// TwinCAT 3 PLC project Master_0000_Allgemein
// ProgramVersion: 3.1.4026.20
// libraries:
//   BASIC, * (OSCAT)
//   Tc2_EtherCAT, * (Beckhoff Automation GmbH)
//   Tc2_MC2, * (Beckhoff Automation GmbH)
//   Tc2_MC2_Drive, * (Beckhoff Automation GmbH)
//   Tc2_NC, * (Beckhoff Automation GmbH)
//   Tc2_Standard, * (Beckhoff Automation GmbH)
//   Tc2_System, * (Beckhoff Automation GmbH)
//   Tc2_Utilities, * (Beckhoff Automation GmbH)
//   Tc3_Database, * (Beckhoff Automation GmbH)
// project tree:
//   0000/ Ablauf_0000.TcPOU, EAs_0000.TcGVL (not stored), GVL_0000.TcGVL (not stored), GVL_Meldungen.TcGVL (not stored), GVL_Visu_0000.TcGVL, Hardware_0000.TcPOU (not stored)
//   1000_Allgemein/ Ablauf_1000.TcPOU (not stored), EAs_1000.TcGVL, GVL_1000.TcGVL, GVL_Visu_1000.TcGVL, Hardware_1000.TcPOU (not stored)
//   3100_Bohraggregat/ Ablauf_3100.TcPOU, EAs_3100.TcGVL (not stored), GVL_3100.TcGVL (not stored), GVL_Visu_3100.TcGVL, Hardware_3100.TcPOU (not stored)
//   3200_Bohraggregat/ Ablauf_3200.TcPOU (not stored), EAs_3200.TcGVL (not stored), GVL_3200.TcGVL, GVL_Visu_3200.TcGVL, Hardware_3200.TcPOU (not stored)
//   3300_Bohraggregat/ Ablauf_3300.TcPOU, EAs_3300.TcGVL, GVL_3300.TcGVL (not stored), GVL_Visu_3300.TcGVL, Hardware_3300.TcPOU
//   3400_Bohraggregat/ Ablauf_3400.TcPOU (not stored), EAs_3400.TcGVL, GVL_3400.TcGVL, GVL_Visu_3400.TcGVL (not stored), Hardware_3400.TcPOU
//   3510_Transport/ Ablauf_3510.TcPOU, EAs_3510.TcGVL (not stored), GVL_3510.TcGVL, GVL_Visu_3510.TcGVL (not stored), Hardware_3510.TcPOU
//   3520_Transport/ Ablauf_3520.TcPOU, EAs_3520.TcGVL (not stored), GVL_3520.TcGVL, GVL_Visu_3520.TcGVL, Hardware_3520.TcPOU (not stored)
//   3530_Niederhalter/ Ablauf_3530.TcPOU, EAs_3530.TcGVL (not stored), GVL_3530.TcGVL, GVL_Visu_3530.TcGVL (not stored), Hardware_3530.TcPOU (not stored)
//   3540_Niederhalter/ Ablauf_3540.TcPOU, EAs_3540.TcGVL, GVL_3540.TcGVL (not stored), GVL_Visu_3540.TcGVL (not stored), Hardware_3540.TcPOU
//   / MAIN.TcPOU (not stored), PlcTask.TcTTO (not stored)
//   SRT_Allgemein/0010_Bausteine_mitDuts/Blink/ GVL_Blink.TcGVL (not stored), PRG_Blink.TcPOU (not stored)
//   SRT_Allgemein/0010_Bausteine_mitDuts/DUTs/ DUT_Visu_SteuerStatus.TcDUT
//   SRT_Allgemein/0010_Bausteine_mitDuts/DUTs/Meldungen/ DUT_Diagnose_1000.TcDUT (not stored), DUT_Diagnose_2000.TcDUT (not stored), DUT_Diagnose_3000.TcDUT, DUT_Diagnose_4000.TcDUT, DUT_Diagnose_5000.TcDUT, DUT_Meldungen_0000.TcDUT, DUT_Diagnose_0000.TcDUT (not stored), DUT_Meldungen_1000.TcDUT, DUT_Meldungen_2000.TcDUT, DUT_Meldungen_3000.TcDUT (not stored), DUT_Meldungen_4000.TcDUT, DUT_Meldungen_5000.TcDUT
//   SRT_Allgemein/0010_Bausteine_mitDuts/DUTs/Rexroth FU/ DUT_Rexroth_FU_PD_IN.TcDUT (not stored), DUT_Rexroth_FU_PD_OUT.TcDUT (not stored), DUT_Rexroth_FU_steuern.TcDUT
//   SRT_Allgemein/0010_Bausteine_mitDuts/DUTs/Safety/ DUT_EL1918_Logic.TcDUT (not stored), E_ModeLanguage.TcDUT (not stored), ST_InfoDataConnection_1904.TcDUT (not stored), ST_InfoDataConnection_1918.TcDUT, ST_InfoDataFB.TcDUT (not stored), ST_InfoDataGroup.TcDUT (not stored)
//   SRT_Allgemein/0010_Bausteine_mitDuts/DUTs/Servo/ DUT_Achse_koppeln.TcDUT (not stored), DUT_Achse_Service.TcDUT, DUT_Achse_Status.TcDUT, DUT_Achse_Steuern.TcDUT (not stored), DUT_Geschwindigkeitsabgleich.TcDUT (not stored), DUT_NC_Kanal.TcDUT (not stored), DUT_PD_InOut_Achsen.TcDUT, DUT_Rexroth_Parameter.TcDUT
//   SRT_Allgemein/0010_Bausteine_mitDuts/DUTs/SEW_Movitrac/COE/ st_COE_Parameter.TcDUT, st_COE_Parameter_Out.TcDUT (not stored)
//   SRT_Allgemein/0010_Bausteine_mitDuts/DUTs/SEW_Movitrac/CSV_BASE/ st_CSV_Database.TcDUT (not stored), st_MaschParameter.TcDUT (not stored)
//   SRT_Allgemein/0010_Bausteine_mitDuts/DUTs/SEW_Movitrac/ DUT_SEW_FU_PD_IN.TcDUT (not stored), DUT_SEW_FU_PD_OUT.TcDUT (not stored), DUT_SEW_FU_Status.TcDUT, DUT_SEW_FU_Steuern.TcDUT (not stored), DUT_SEW_FU_Visu.TcDUT, DUT_SEW_Para.TcDUT (not stored)
//   SRT_Allgemein/0010_Bausteine_mitDuts/DUTs/Ventil/ DUT_Ventil_para.TcDUT, DUT_Ventil_sps.TcDUT (not stored), DUT_Ventil_VISU.TcDUT, DUT_VorZur_visu.TcDUT (not stored)
//   SRT_Allgemein/0010_Bausteine_mitDuts/POUs/ FB_Achs_Freigabe.TcPOU, FB_Anst_Vakuum.TcPOU (not stored), FB_Automatik.TcPOU, FB_Belegt.TcPOU, FB_Bereichsueberwachung.TcPOU, FB_FuStart_Fraese.TcPOU (not stored), FB_FU_Rexroth.TcPOU, FB_inRange.TcPOU (not stored), FB_Kollision.TcPOU (not stored), FB_Messachse_EL3051.TcPOU, FB_Messachse_EL5151.TcPOU (not stored), FB_Messauswertung_Hysterese.TcPOU (not stored), FB_normieren.TcPOU (not stored), FB_PneuPosition.TcPOU (not stored), FB_Schutztuer_mitBremsentest.TcPOU, FB_Toggle_Anforderung.TcPOU (not stored), FB_Toogle.TcPOU (not stored), FB_Transport.TcPOU (not stored), FB_Umrechnung.TcPOU (not stored), FB_Ventil.TcPOU, FB_Ventil_V2.TcPOU, FC_Bereichsueberwachung.TcPOU, FC_InRange.TcPOU, Func_InRange.TcPOU (not stored), IBN_Huettenhoelscher.TcPOU (not stored)
//   SRT_Allgemein/0010_Bausteine_mitDuts/POUs/FU_SEW/Movi_B/ FB_SEW_MOVITRAC.TcPOU, FB_SEW_MOVITRAC_CoE.TcPOU (not stored)
//   SRT_Allgemein/0010_Bausteine_mitDuts/POUs/FU_SEW/Movi_C/ FB_SEW_MOVITRAC_C_COE.TcPOU, FB_SEW_MOVITRAC_C_COE_18000Umin.TcPOU (not stored)
//   SRT_Allgemein/0010_Bausteine_mitDuts/POUs/FU_SEW/sub/CoE/ fb_CoeDataRead.TcPOU (not stored), fb_CoeDataWrite.TcPOU (not stored)
//   SRT_Allgemein/0010_Bausteine_mitDuts/POUs/FU_SEW/sub/CSV Read_Write/ fb_CSVBaseRead.TcPOU, fb_CSVBaseWrite.TcPOU (not stored), fb_OrdnerErstellen.TcPOU, fb_Parameter_CSV.TcPOU
//   SRT_Allgemein/0010_Bausteine_mitDuts/POUs/FU_SEW/sub/ FB_SEW_CoE.TcPOU (not stored)
//   SRT_Allgemein/0010_Bausteine_mitDuts/POUs/Safety/ FB_InfoConnection_1904.TcPOU (not stored), FB_InfoConnection_1918.TcPOU, FB_InfoEStop.TcPOU, FB_InfoGroup.TcPOU (not stored)
//   SRT_Allgemein/0010_Bausteine_mitDuts/POUs/Servos_NC/ FB_Achse_NC_PTP_Beckhoff.TcPOU (not stored), FB_Achse_NC_PTP_Master_Slave_v2.TcPOU, FB_Achse_NC_PTP_V3.TcPOU, FB_Achse_NC_PTP_V4.TcPOU, FB_Achse_NC_PTP_V4_1.TcPOU (not stored), FB_Achse_NC_PTP_V4_2.TcPOU, FB_Achse_NC_PTP_Velo.TcPOU (not stored), FB_MasterSlaveSpeedControl.TcPOU, FB_Nc_Kanal.TcPOU, Rexroth_Servo_Modulo.TcPOU (not stored)
//   SRT_Allgemein/0010_Bausteine_mitDuts/POUs/Zaehler/ FB_Laufzeit.TcPOU, FB_SpindelInBearbeitung.TcPOU
//   SRT_Allgemein/Bus/ Busdiagnose.TcPOU, DUT_Busdiagnose.TcDUT, DUT_Busdiagnose_Daten.TcDUT (not stored), GVL_Busdiagnose.TcGVL (not stored)
// real-time tasks:
//   TASK PlcTask: cycle T#10ms, priority 20, ADS port 350
// motion (NC):
//   TASK NC-Task 1 SAF: cycle T#2ms, priority 4, ADS port 501
//   TASK NC-Task 1 SVB: cycle T#10ms, priority 8, ADS port 511
//   AXIS =3100+FS2-11M1 (X-Achse) (id 1)
//     OtherSettings: AllowMotionCmdToSlave=true
//     encoder EncType=19
//       EncPara: MaxCount=#xffffffff
//     drive DrvType=16
//       DrvPara: MaxCount=#xffffffff
//         Analog: TorqueSetpointScale=10, ScaleFactorActTorque=0.1
//         TimeComp: TaskDelayCycles=1
//     controller CtrType=1
//       CtrPara: PriorControlFactor=1
//         Observer: BandWidth=20
//   AXIS =3100+FS2-12M1 (Y-Achse) (id 2)
//     OtherSettings: AllowMotionCmdToSlave=true
//     encoder EncType=19
//       EncPara: MaxCount=#xffffffff
//     drive DrvType=16
//       DrvPara: MaxCount=#xffffffff
//         Analog: TorqueSetpointScale=10, ScaleFactorActTorque=0.1
//         TimeComp: TaskDelayCycles=1
//     controller CtrType=1
//       CtrPara: PriorControlFactor=1
//         Observer: BandWidth=20
//   AXIS =3100+FS2-13M1 (Z-Achse) (id 3)
//     OtherSettings: AllowMotionCmdToSlave=true
//     encoder EncType=19
//       EncPara: MaxCount=#xffffffff
//     drive DrvType=16
//       DrvPara: MaxCount=#xffffffff
//         Analog: TorqueSetpointScale=10, ScaleFactorActTorque=0.1
//         TimeComp: TaskDelayCycles=1
//     controller CtrType=1
//       CtrPara: PriorControlFactor=1
//         Observer: BandWidth=20
//   AXIS =3200+FS2-11M1 (X-Achse) (id 4)
//     OtherSettings: AllowMotionCmdToSlave=true
//     encoder EncType=19
//       EncPara: MaxCount=#xffffffff
//     drive DrvType=16
//       DrvPara: MaxCount=#xffffffff
//         Analog: TorqueSetpointScale=10, ScaleFactorActTorque=0.1
//         TimeComp: TaskDelayCycles=1
//     controller CtrType=1
//       CtrPara: PriorControlFactor=1
//         Observer: BandWidth=20
//   AXIS =3200+FS2-12M1 (Y-Achse) (id 5)
//     OtherSettings: AllowMotionCmdToSlave=true
//     encoder EncType=19
//       EncPara: MaxCount=#xffffffff
//     drive DrvType=16
//       DrvPara: MaxCount=#xffffffff
//         Analog: TorqueSetpointScale=10, ScaleFactorActTorque=0.1
//         TimeComp: TaskDelayCycles=1
//     controller CtrType=1
//       CtrPara: PriorControlFactor=1
//         Observer: BandWidth=20
//   AXIS =3200+FS2-13M1 (Z-Achse) (id 6)
//     OtherSettings: AllowMotionCmdToSlave=true
//     encoder EncType=19
//       EncPara: MaxCount=#xffffffff
//     drive DrvType=16
//       DrvPara: MaxCount=#xffffffff
//         Analog: TorqueSetpointScale=10, ScaleFactorActTorque=0.1
//         TimeComp: TaskDelayCycles=1
//     controller CtrType=1
//       CtrPara: PriorControlFactor=1
//         Observer: BandWidth=20
//   AXIS =3300+FS2-11M1 (X-Achse) (id 7)
//     OtherSettings: AllowMotionCmdToSlave=true
//     encoder EncType=19
//       EncPara: MaxCount=#xffffffff
//     drive DrvType=16
//       DrvPara: MaxCount=#xffffffff
//         Analog: TorqueSetpointScale=10, ScaleFactorActTorque=0.1
//         TimeComp: TaskDelayCycles=1
//     controller CtrType=1
//       CtrPara: PriorControlFactor=1
//         Observer: BandWidth=20
//   AXIS =3300+FS2-12M1 (Y-Achse) (id 8)
//     OtherSettings: AllowMotionCmdToSlave=true
//     encoder EncType=19
//       EncPara: MaxCount=#xffffffff
//     drive DrvType=16
//       DrvPara: MaxCount=#xffffffff
//         Analog: TorqueSetpointScale=10, ScaleFactorActTorque=0.1
//         TimeComp: TaskDelayCycles=1
//     controller CtrType=1
//       CtrPara: PriorControlFactor=1
//         Observer: BandWidth=20
//   AXIS =3400+FS2-11M1 (X-Achse) (id 9)
//     OtherSettings: AllowMotionCmdToSlave=true
//     encoder EncType=19
//       EncPara: MaxCount=#xffffffff
//     drive DrvType=16
//       DrvPara: MaxCount=#xffffffff
//         Analog: TorqueSetpointScale=10, ScaleFactorActTorque=0.1
//         TimeComp: TaskDelayCycles=1
//     controller CtrType=1
//       CtrPara: PriorControlFactor=1
//         Observer: BandWidth=20
//   AXIS =3400+FS2-12M1 (Y-Achse) (id 10)
//     OtherSettings: AllowMotionCmdToSlave=true
//     encoder EncType=19
//       EncPara: MaxCount=#xffffffff
//     drive DrvType=16
//       DrvPara: MaxCount=#xffffffff
//         Analog: TorqueSetpointScale=10, ScaleFactorActTorque=0.1
//         TimeComp: TaskDelayCycles=1
//     controller CtrType=1
//       CtrPara: PriorControlFactor=1
//         Observer: BandWidth=20
//   AXIS =3520+FS2-11M1 (Y-Achse) (id 11)
//     OtherSettings: AllowMotionCmdToSlave=true
//     encoder EncType=19
//       EncPara: MaxCount=#xffffffff
//     drive DrvType=16
//       DrvPara: MaxCount=#xffffffff
//         Analog: TorqueSetpointScale=10, ScaleFactorActTorque=0.1
//         TimeComp: TaskDelayCycles=1
//     controller CtrType=1
//       CtrPara: PriorControlFactor=1
//         Observer: BandWidth=20
//   AXIS =3540+FS2-11M1 (Y-Achse) (id 12)
//     OtherSettings: AllowMotionCmdToSlave=true
//     encoder EncType=19
//       EncPara: MaxCount=#xffffffff
//     drive DrvType=16
//       DrvPara: MaxCount=#xffffffff
//         Analog: TorqueSetpointScale=10, ScaleFactorActTorque=0.1
//         TimeComp: TaskDelayCycles=1
//     controller CtrType=1
//       CtrPara: PriorControlFactor=1
//         Observer: BandWidth=20
// I/O:
//   DEVICE Gerät 1 (EtherCAT), AmsNetId 169.254.68.135.2.1
//     +FS1-3K1 (BK1120) [EK1100 EtherCAT-Koppler (2A E-Bus)]
//       +FS1-3K2 (EL6070-0033) [EL6070-0033 1K. Licence-Key-Klemme, individuelle Lizenzen]
//       +FS1-3K3 (EL1918) [EL1918, 8K. Safety Eingang 24V, TwinSAFE]
//         modules: Module 1 (FSOE), Module 2 (FSLOGIC)
//       +FS1-3K4 (EL2904) [EL2904, 4 K. Safety Ausgang 24V, 0.5A, TwinSAFE]
//         modules: Module 1 (FSOES), Module 2 (DO)
//       +FS1-3K5 (EL1809)
//       +FS1-3K6 (EL2809)
//       +FS1-3A1 (EL9011)
//     +K110-1K1 (BK1120)
//     =3100+FS2-16T1 (Bohraggr Schlosskastenfräser) [MOVI-C MOVITRAC]
//       modules: Module 1 (Standard 16 PD)
//     =3100+FS2-17T1 (Bohraggr Vorbohren) [MOVI-C MOVITRAC]
//       modules: Module 1 (Standard 16 PD)
//     =3100+FS2-18T1 (Bohraggr Stulpfräser) [MOVI-C MOVITRAC]
//       modules: Module 1 (Standard 16 PD)
//     =3200+FS2-16T1 (Bohraggr Stufenbohrer) [MOVI-C MOVITRAC]
//       modules: Module 1 (Standard 16 PD)
//     =3200+FS2-17T1 (Bohraggr Stulpfräser) [MOVI-C MOVITRAC]
//       modules: Module 1 (Standard 16 PD)
//     =3300+FS2-16T1 (Bohraggr Schlüsselloch unten) [MOVI-C MOVITRAC]
//       modules: Module 1 (Standard 16 PD)
//     =3400+FS2-16T1 (Bohraggr Schlüsselloch oben) [MOVI-C MOVITRAC]
//       modules: Module 1 (Standard 16 PD)
//     =3510+FS2-6T1 (Transport Schlossseite X-Achse) [MOVI-C MOVITRAC]
//       modules: Module 1 (Standard 16 PD)
//     =3520+FS2-6T1 (Transport Bandseite X-Achse)
//     =0300+FS2-13T1 [MOVI-C MOVIDRIVE CiA402]
//       modules: =3100+FS2-11M1 (X-Achse), Module 2 (FSoE empty), =3100+FS2-12M1 (Y-Achse), Module 4 (FSoE empty)
//     =0300+FS2-14T1 [MOVI-C MOVIDRIVE CiA402]
//       modules: =3100+FS2-14M1 (Z-Achse), Module 2 (FSoE empty), =3200+FS2-11M1 (X-Achse), Module 4 (FSoE empty)
//     =0300+FS2-15T1 [MOVI-C MOVIDRIVE CiA402]
//       modules: =3200+FS2-12M1 (Y-Achse), Module 2 (FSoE empty), =3200+FS2-13M1 (Z-Achse), Module 4 (FSoE empty)
//     =0300+FS2-16T1 [MOVI-C MOVIDRIVE CiA402]
//       modules: =3300+FS2-11M1 (X-Achse), Module 2 (FSoE empty), =3300+FS2-12M1 (Y-Achse), Module 4 (FSoE empty)
//     =0300+FS2-17T1 [MOVI-C MOVIDRIVE CiA402]
//       modules: =3400+FS2-11M1 (X-Achse), Module 2 (FSoE empty), =3400+FS2-12M1 (Y-Achse), Module 4 (FSoE empty)
//     =0300+FS2-18T1 [MOVI-C MOVIDRIVE CiA402]
//       modules: =3520+FS2-11M1 (Y-Achse Riemenförderer), Module 2 (FSoE empty), =3540+FS2-11M1 (Y-Achse), Module 4 (FSoE empty)
// variable links:
//   (this object) <-> Device 1 (EtherCAT)/=0300+FS2-13T1
//     Drive/Inputs/In/nDataIn3[0] <-> =3100+FS2-11M1 (X-Achse)/Inputs/Torque actual value
//     Drive/Inputs/In/nDcOutputTime <-> InfoData/DcOutputShift
//     Drive/Inputs/In/nState1 <-> =3100+FS2-11M1 (X-Achse)/Inputs/Status word
//     Drive/Inputs/In/nState2 <-> =3100+FS2-11M1 (X-Achse)/Inputs/Status word @bit 8
//     Drive/Inputs/In/nState4 @bit 1 <-> WcState/InputToggle
//     Drive/Inputs/In/nState4 <-> WcState/WcState
//     Drive/Inputs/In/nState5 <-> =3100+FS2-11M1 (X-Achse)/Inputs/Modes of operation display
//     Drive/Outputs/Out/nCtrl1 <-> =3100+FS2-11M1 (X-Achse)/Outputs/Control word
//     Drive/Outputs/Out/nCtrl2 <-> =3100+FS2-11M1 (X-Achse)/Outputs/Control word @bit 8
//     Drive/Outputs/Out/nCtrl5 <-> =3100+FS2-11M1 (X-Achse)/Outputs/Modes of operation
//     Drive/Outputs/Out/nDataOut1 <-> =3100+FS2-11M1 (X-Achse)/Outputs/Target position
//     Drive/Outputs/Out/nDataOut2 <-> =3100+FS2-11M1 (X-Achse)/Outputs/Target velocity
//     Drive/Outputs/Out/nDataOut4[0] <-> =3100+FS2-11M1 (X-Achse)/Outputs/Target torque
//     Enc/Inputs/In/nDataIn1 <-> =3100+FS2-11M1 (X-Achse)/Inputs/Position actual value
//     Enc/Inputs/In/nDcInputTime <-> InfoData/DcInputShift
//     Enc/Inputs/In/nState4 @bit 1 <-> WcState/InputToggle
//     Enc/Inputs/In/nState4 <-> WcState/WcState
//     Drive/Inputs/In/nDataIn3[0] <-> =3100+FS2-12M1 (Y-Achse)/Inputs/Torque actual value
//     Drive/Inputs/In/nState1 <-> =3100+FS2-12M1 (Y-Achse)/Inputs/Status word
//     Drive/Inputs/In/nState2 <-> =3100+FS2-12M1 (Y-Achse)/Inputs/Status word @bit 8
//     Drive/Inputs/In/nState5 <-> =3100+FS2-12M1 (Y-Achse)/Inputs/Modes of operation display
//     Drive/Outputs/Out/nCtrl1 <-> =3100+FS2-12M1 (Y-Achse)/Outputs/Control word
//     Drive/Outputs/Out/nCtrl2 <-> =3100+FS2-12M1 (Y-Achse)/Outputs/Control word @bit 8
//     Drive/Outputs/Out/nCtrl5 <-> =3100+FS2-12M1 (Y-Achse)/Outputs/Modes of operation
//     Drive/Outputs/Out/nDataOut1 <-> =3100+FS2-12M1 (Y-Achse)/Outputs/Target position
//     Drive/Outputs/Out/nDataOut2 <-> =3100+FS2-12M1 (Y-Achse)/Outputs/Target velocity
//     Drive/Outputs/Out/nDataOut4[0] <-> =3100+FS2-12M1 (Y-Achse)/Outputs/Target torque
//     Enc/Inputs/In/nDataIn1 <-> =3100+FS2-12M1 (Y-Achse)/Inputs/Position actual value
//   (this object) <-> Device 1 (EtherCAT)/=0300+FS2-14T1
//     Drive/Inputs/In/nDataIn3[0] <-> =3100+FS2-14M1 (Z-Achse)/Inputs/Torque actual value
//     Drive/Inputs/In/nDcOutputTime <-> InfoData/DcOutputShift
//     Drive/Inputs/In/nState1 <-> =3100+FS2-14M1 (Z-Achse)/Inputs/Status word
//     Drive/Inputs/In/nState2 <-> =3100+FS2-14M1 (Z-Achse)/Inputs/Status word @bit 8
//     Drive/Inputs/In/nState4 @bit 1 <-> WcState/InputToggle
//     Drive/Inputs/In/nState4 <-> WcState/WcState
//     Drive/Inputs/In/nState5 <-> =3100+FS2-14M1 (Z-Achse)/Inputs/Modes of operation display
//     Drive/Outputs/Out/nCtrl1 <-> =3100+FS2-14M1 (Z-Achse)/Outputs/Control word
//     Drive/Outputs/Out/nCtrl2 <-> =3100+FS2-14M1 (Z-Achse)/Outputs/Control word @bit 8
//     Drive/Outputs/Out/nCtrl5 <-> =3100+FS2-14M1 (Z-Achse)/Outputs/Modes of operation
//     Drive/Outputs/Out/nDataOut1 <-> =3100+FS2-14M1 (Z-Achse)/Outputs/Target position
//     Drive/Outputs/Out/nDataOut2 <-> =3100+FS2-14M1 (Z-Achse)/Outputs/Target velocity
//     Drive/Outputs/Out/nDataOut4[0] <-> =3100+FS2-14M1 (Z-Achse)/Outputs/Target torque
//     Enc/Inputs/In/nDataIn1 <-> =3100+FS2-14M1 (Z-Achse)/Inputs/Position actual value
//     Enc/Inputs/In/nDcInputTime <-> InfoData/DcInputShift
//     Enc/Inputs/In/nState4 @bit 1 <-> WcState/InputToggle
//     Enc/Inputs/In/nState4 <-> WcState/WcState
//     Drive/Inputs/In/nDataIn3[0] <-> =3200+FS2-11M1 (X-Achse)/Inputs/Torque actual value
//     Drive/Inputs/In/nState1 <-> =3200+FS2-11M1 (X-Achse)/Inputs/Status word
//     Drive/Inputs/In/nState2 <-> =3200+FS2-11M1 (X-Achse)/Inputs/Status word @bit 8
//     Drive/Inputs/In/nState5 <-> =3200+FS2-11M1 (X-Achse)/Inputs/Modes of operation display
//     Drive/Outputs/Out/nCtrl1 <-> =3200+FS2-11M1 (X-Achse)/Outputs/Control word
//     Drive/Outputs/Out/nCtrl2 <-> =3200+FS2-11M1 (X-Achse)/Outputs/Control word @bit 8
//     Drive/Outputs/Out/nCtrl5 <-> =3200+FS2-11M1 (X-Achse)/Outputs/Modes of operation
//     Drive/Outputs/Out/nDataOut1 <-> =3200+FS2-11M1 (X-Achse)/Outputs/Target position
//     Drive/Outputs/Out/nDataOut2 <-> =3200+FS2-11M1 (X-Achse)/Outputs/Target velocity
//     Drive/Outputs/Out/nDataOut4[0] <-> =3200+FS2-11M1 (X-Achse)/Outputs/Target torque
//     Enc/Inputs/In/nDataIn1 <-> =3200+FS2-11M1 (X-Achse)/Inputs/Position actual value
//   (this object) <-> Device 1 (EtherCAT)/=0300+FS2-15T1
//     Drive/Inputs/In/nDataIn3[0] <-> =3200+FS2-12M1 (Y-Achse)/Inputs/Torque actual value
//     Drive/Inputs/In/nDcOutputTime <-> InfoData/DcOutputShift
//     Drive/Inputs/In/nState1 <-> =3200+FS2-12M1 (Y-Achse)/Inputs/Status word
//     Drive/Inputs/In/nState2 <-> =3200+FS2-12M1 (Y-Achse)/Inputs/Status word @bit 8
//     Drive/Inputs/In/nState4 @bit 1 <-> WcState/InputToggle
//     Drive/Inputs/In/nState4 <-> WcState/WcState
//     Drive/Inputs/In/nState5 <-> =3200+FS2-12M1 (Y-Achse)/Inputs/Modes of operation display
//     Drive/Outputs/Out/nCtrl1 <-> =3200+FS2-12M1 (Y-Achse)/Outputs/Control word
//     Drive/Outputs/Out/nCtrl2 <-> =3200+FS2-12M1 (Y-Achse)/Outputs/Control word @bit 8
//     Drive/Outputs/Out/nCtrl5 <-> =3200+FS2-12M1 (Y-Achse)/Outputs/Modes of operation
//     Drive/Outputs/Out/nDataOut1 <-> =3200+FS2-12M1 (Y-Achse)/Outputs/Target position
//     Drive/Outputs/Out/nDataOut2 <-> =3200+FS2-12M1 (Y-Achse)/Outputs/Target velocity
//     Drive/Outputs/Out/nDataOut4[0] <-> =3200+FS2-12M1 (Y-Achse)/Outputs/Target torque
//     Enc/Inputs/In/nDataIn1 <-> =3200+FS2-12M1 (Y-Achse)/Inputs/Position actual value
//     Enc/Inputs/In/nDcInputTime <-> InfoData/DcInputShift
//     Enc/Inputs/In/nState4 @bit 1 <-> WcState/InputToggle
//     Enc/Inputs/In/nState4 <-> WcState/WcState
//     Drive/Inputs/In/nDataIn3[0] <-> =3200+FS2-13M1 (Z-Achse)/Inputs/Torque actual value
//     Drive/Inputs/In/nState1 <-> =3200+FS2-13M1 (Z-Achse)/Inputs/Status word
//     Drive/Inputs/In/nState2 <-> =3200+FS2-13M1 (Z-Achse)/Inputs/Status word @bit 8
//     Drive/Inputs/In/nState5 <-> =3200+FS2-13M1 (Z-Achse)/Inputs/Modes of operation display
//     Drive/Outputs/Out/nCtrl1 <-> =3200+FS2-13M1 (Z-Achse)/Outputs/Control word
//     Drive/Outputs/Out/nCtrl2 <-> =3200+FS2-13M1 (Z-Achse)/Outputs/Control word @bit 8
//     Drive/Outputs/Out/nCtrl5 <-> =3200+FS2-13M1 (Z-Achse)/Outputs/Modes of operation
//     Drive/Outputs/Out/nDataOut1 <-> =3200+FS2-13M1 (Z-Achse)/Outputs/Target position
//     Drive/Outputs/Out/nDataOut2 <-> =3200+FS2-13M1 (Z-Achse)/Outputs/Target velocity
//     Drive/Outputs/Out/nDataOut4[0] <-> =3200+FS2-13M1 (Z-Achse)/Outputs/Target torque
//     Enc/Inputs/In/nDataIn1 <-> =3200+FS2-13M1 (Z-Achse)/Inputs/Position actual value
//   (this object) <-> Device 1 (EtherCAT)/=0300+FS2-16T1
//     Drive/Inputs/In/nDataIn3[0] <-> =3300+FS2-11M1 (X-Achse)/Inputs/Torque actual value
//     Drive/Inputs/In/nDcOutputTime <-> InfoData/DcOutputShift
//     Drive/Inputs/In/nState1 <-> =3300+FS2-11M1 (X-Achse)/Inputs/Status word
//     Drive/Inputs/In/nState2 <-> =3300+FS2-11M1 (X-Achse)/Inputs/Status word @bit 8
//     Drive/Inputs/In/nState4 @bit 1 <-> WcState/InputToggle
//     Drive/Inputs/In/nState4 <-> WcState/WcState
//     Drive/Inputs/In/nState5 <-> =3300+FS2-11M1 (X-Achse)/Inputs/Modes of operation display
//     Drive/Outputs/Out/nCtrl1 <-> =3300+FS2-11M1 (X-Achse)/Outputs/Control word
//     Drive/Outputs/Out/nCtrl2 <-> =3300+FS2-11M1 (X-Achse)/Outputs/Control word @bit 8
//     Drive/Outputs/Out/nCtrl5 <-> =3300+FS2-11M1 (X-Achse)/Outputs/Modes of operation
//     Drive/Outputs/Out/nDataOut1 <-> =3300+FS2-11M1 (X-Achse)/Outputs/Target position
//     Drive/Outputs/Out/nDataOut2 <-> =3300+FS2-11M1 (X-Achse)/Outputs/Target velocity
//     Drive/Outputs/Out/nDataOut4[0] <-> =3300+FS2-11M1 (X-Achse)/Outputs/Target torque
//     Enc/Inputs/In/nDataIn1 <-> =3300+FS2-11M1 (X-Achse)/Inputs/Position actual value
//     Enc/Inputs/In/nDcInputTime <-> InfoData/DcInputShift
//     Enc/Inputs/In/nState4 @bit 1 <-> WcState/InputToggle
//     Enc/Inputs/In/nState4 <-> WcState/WcState
//     Drive/Inputs/In/nDataIn3[0] <-> =3300+FS2-12M1 (Y-Achse)/Inputs/Torque actual value
//     Drive/Inputs/In/nState1 <-> =3300+FS2-12M1 (Y-Achse)/Inputs/Status word
//     Drive/Inputs/In/nState2 <-> =3300+FS2-12M1 (Y-Achse)/Inputs/Status word @bit 8
//     Drive/Inputs/In/nState5 <-> =3300+FS2-12M1 (Y-Achse)/Inputs/Modes of operation display
//     Drive/Outputs/Out/nCtrl1 <-> =3300+FS2-12M1 (Y-Achse)/Outputs/Control word
//     Drive/Outputs/Out/nCtrl2 <-> =3300+FS2-12M1 (Y-Achse)/Outputs/Control word @bit 8
//     Drive/Outputs/Out/nCtrl5 <-> =3300+FS2-12M1 (Y-Achse)/Outputs/Modes of operation
//     Drive/Outputs/Out/nDataOut1 <-> =3300+FS2-12M1 (Y-Achse)/Outputs/Target position
//     Drive/Outputs/Out/nDataOut2 <-> =3300+FS2-12M1 (Y-Achse)/Outputs/Target velocity
//     Drive/Outputs/Out/nDataOut4[0] <-> =3300+FS2-12M1 (Y-Achse)/Outputs/Target torque
//     Enc/Inputs/In/nDataIn1 <-> =3300+FS2-12M1 (Y-Achse)/Inputs/Position actual value
//   (this object) <-> Device 1 (EtherCAT)/=0300+FS2-17T1
//     Drive/Inputs/In/nDataIn3[0] <-> =3400+FS2-11M1 (X-Achse)/Inputs/Torque actual value
//     Drive/Inputs/In/nDcOutputTime <-> InfoData/DcOutputShift
//     Drive/Inputs/In/nState1 <-> =3400+FS2-11M1 (X-Achse)/Inputs/Status word
//     Drive/Inputs/In/nState2 <-> =3400+FS2-11M1 (X-Achse)/Inputs/Status word @bit 8
//     Drive/Inputs/In/nState4 @bit 1 <-> WcState/InputToggle
//     Drive/Inputs/In/nState4 <-> WcState/WcState
//     Drive/Inputs/In/nState5 <-> =3400+FS2-11M1 (X-Achse)/Inputs/Modes of operation display
//     Drive/Outputs/Out/nCtrl1 <-> =3400+FS2-11M1 (X-Achse)/Outputs/Control word
//     Drive/Outputs/Out/nCtrl2 <-> =3400+FS2-11M1 (X-Achse)/Outputs/Control word @bit 8
//     Drive/Outputs/Out/nCtrl5 <-> =3400+FS2-11M1 (X-Achse)/Outputs/Modes of operation
//     Drive/Outputs/Out/nDataOut1 <-> =3400+FS2-11M1 (X-Achse)/Outputs/Target position
//     Drive/Outputs/Out/nDataOut2 <-> =3400+FS2-11M1 (X-Achse)/Outputs/Target velocity
//     Drive/Outputs/Out/nDataOut4[0] <-> =3400+FS2-11M1 (X-Achse)/Outputs/Target torque
//     Enc/Inputs/In/nDataIn1 <-> =3400+FS2-11M1 (X-Achse)/Inputs/Position actual value
//     Enc/Inputs/In/nDcInputTime <-> InfoData/DcInputShift
//     Enc/Inputs/In/nState4 @bit 1 <-> WcState/InputToggle
//     Enc/Inputs/In/nState4 <-> WcState/WcState
//     Drive/Inputs/In/nDataIn3[0] <-> =3400+FS2-12M1 (Y-Achse)/Inputs/Torque actual value
//     Drive/Inputs/In/nState1 <-> =3400+FS2-12M1 (Y-Achse)/Inputs/Status word
//     Drive/Inputs/In/nState2 <-> =3400+FS2-12M1 (Y-Achse)/Inputs/Status word @bit 8
//     Drive/Inputs/In/nState5 <-> =3400+FS2-12M1 (Y-Achse)/Inputs/Modes of operation display
//     Drive/Outputs/Out/nCtrl1 <-> =3400+FS2-12M1 (Y-Achse)/Outputs/Control word
//     Drive/Outputs/Out/nCtrl2 <-> =3400+FS2-12M1 (Y-Achse)/Outputs/Control word @bit 8
//     Drive/Outputs/Out/nCtrl5 <-> =3400+FS2-12M1 (Y-Achse)/Outputs/Modes of operation
//     Drive/Outputs/Out/nDataOut1 <-> =3400+FS2-12M1 (Y-Achse)/Outputs/Target position
//     Drive/Outputs/Out/nDataOut2 <-> =3400+FS2-12M1 (Y-Achse)/Outputs/Target velocity
//     Drive/Outputs/Out/nDataOut4[0] <-> =3400+FS2-12M1 (Y-Achse)/Outputs/Target torque
//     Enc/Inputs/In/nDataIn1 <-> =3400+FS2-12M1 (Y-Achse)/Inputs/Position actual value
//   (this object) <-> Device 1 (EtherCAT)/=0300+FS2-18T1
//     Drive/Inputs/In/nDataIn3[0] <-> =3520+FS2-11M1 (Y-Achse Riemenförderer)/Inputs/Torque actual value
//     Drive/Inputs/In/nDcOutputTime <-> InfoData/DcOutputShift
//     Drive/Inputs/In/nState1 <-> =3520+FS2-11M1 (Y-Achse Riemenförderer)/Inputs/Status word
//     Drive/Inputs/In/nState2 <-> =3520+FS2-11M1 (Y-Achse Riemenförderer)/Inputs/Status word @bit 8
//     Drive/Inputs/In/nState4 @bit 1 <-> WcState/InputToggle
//     Drive/Inputs/In/nState4 <-> WcState/WcState
//     Drive/Inputs/In/nState5 <-> =3520+FS2-11M1 (Y-Achse Riemenförderer)/Inputs/Modes of operation display
//     Drive/Outputs/Out/nCtrl1 <-> =3520+FS2-11M1 (Y-Achse Riemenförderer)/Outputs/Control word
//     Drive/Outputs/Out/nCtrl2 <-> =3520+FS2-11M1 (Y-Achse Riemenförderer)/Outputs/Control word @bit 8
//     Drive/Outputs/Out/nCtrl5 <-> =3520+FS2-11M1 (Y-Achse Riemenförderer)/Outputs/Modes of operation
//     Drive/Outputs/Out/nDataOut1 <-> =3520+FS2-11M1 (Y-Achse Riemenförderer)/Outputs/Target position
//     Drive/Outputs/Out/nDataOut2 <-> =3520+FS2-11M1 (Y-Achse Riemenförderer)/Outputs/Target velocity
//     Drive/Outputs/Out/nDataOut4[0] <-> =3520+FS2-11M1 (Y-Achse Riemenförderer)/Outputs/Target torque
//     Enc/Inputs/In/nDataIn1 <-> =3520+FS2-11M1 (Y-Achse Riemenförderer)/Inputs/Position actual value
//     Enc/Inputs/In/nDcInputTime <-> InfoData/DcInputShift
//     Enc/Inputs/In/nState4 @bit 1 <-> WcState/InputToggle
//     Enc/Inputs/In/nState4 <-> WcState/WcState
//     Drive/Inputs/In/nDataIn3[0] <-> =3540+FS2-11M1 (Y-Achse)/Inputs/Torque actual value
//     Drive/Inputs/In/nState1 <-> =3540+FS2-11M1 (Y-Achse)/Inputs/Status word
//     Drive/Inputs/In/nState2 <-> =3540+FS2-11M1 (Y-Achse)/Inputs/Status word @bit 8
//     Drive/Inputs/In/nState5 <-> =3540+FS2-11M1 (Y-Achse)/Inputs/Modes of operation display
//     Drive/Outputs/Out/nCtrl1 <-> =3540+FS2-11M1 (Y-Achse)/Outputs/Control word
//     Drive/Outputs/Out/nCtrl2 <-> =3540+FS2-11M1 (Y-Achse)/Outputs/Control word @bit 8
//     Drive/Outputs/Out/nCtrl5 <-> =3540+FS2-11M1 (Y-Achse)/Outputs/Modes of operation
//     Drive/Outputs/Out/nDataOut1 <-> =3540+FS2-11M1 (Y-Achse)/Outputs/Target position
//     Drive/Outputs/Out/nDataOut2 <-> =3540+FS2-11M1 (Y-Achse)/Outputs/Target velocity
//     Drive/Outputs/Out/nDataOut4[0] <-> =3540+FS2-11M1 (Y-Achse)/Outputs/Target torque
//     Enc/Inputs/In/nDataIn1 <-> =3540+FS2-11M1 (Y-Achse)/Inputs/Position actual value
//   (this object) <-> Device 1 (EtherCAT)/+FS1-3K1 (BK1120)/+FS1-3K5 (EL1809)
//     PlcTask Inputs/EAs_0000.e_FR_0101_Schaltschranktuer_ist_zu_und_Klimageraet_ist_Betriebsbereit <-> Channel 1/Input
//     PlcTask Inputs/EAs_0000.e_FR_0300_SEW_Bremswiderstand_Versorgungsmodul_ist_OK <-> Channel 13/Input
//     PlcTask Inputs/EAs_0000.e_FR_0400_Schaltschrank_24V_Lastueberwachung_ist_OK <-> Channel 2/Input
//     PlcTask Inputs/EAs_0000.e_FR_0600_Rueckmeldung_von_Safety_Freigabekreis_3 <-> Channel 3/Input
//     PlcTask Inputs/EAs_0000.e_FR_0800_24V_UPS_Versorgung_ist_OK_und_zu_80_geladen <-> Channel 4/Input
//     PlcTask Inputs/EAs_0000.e_FS1_3K5_Channel_14 <-> Channel 14/Input
//     PlcTask Inputs/EAs_0000.e_FS1_3K5_Channel_15 <-> Channel 15/Input
//     PlcTask Inputs/EAs_0000.e_FS1_3K5_Channel_16 <-> Channel 16/Input
//     PlcTask Inputs/EAs_1000.e_FR_1000_Allgemein_Druckluft_OK <-> Channel 5/Input
//     PlcTask Inputs/EAs_3100.e_FR_3100_Bohraggregat_1_Schlosskastenfraeser_Stillstandserkennung_Motor_steht <-> Channel 6/Input
//     PlcTask Inputs/EAs_3100.e_FR_3100_Bohraggregat_2_Vorbohren_Stillstandserkennung_Motor_steht <-> Channel 7/Input
//     PlcTask Inputs/EAs_3100.e_FR_3100_Bohraggregat_3_Stulpfraeser_Stillstandserkennung_Motor_steht <-> Channel 8/Input
//     PlcTask Inputs/EAs_3200.e_FR_3200_Bohraggregat_5_Stulpfraeser_Stillstandserkennung_Motor_steht <-> Channel 10/Input
//     PlcTask Inputs/EAs_3200.e_FR_3200_Bohraggregat_4_Stufenbohrer_Stillstandserkennung_Motor_steht <-> Channel 9/Input
//     PlcTask Inputs/EAs_3300.e_FR_3300_Bohraggregat_6_Schluesselloch_unten_Stillstandserkennung_Motor_steht <-> Channel 11/Input
//     PlcTask Inputs/EAs_3400.e_FR_3400_Bohraggregat_7_Schluesselloch_oben_Stillstandserkennung_Motor_steht <-> Channel 12/Input
//   (this object) <-> Device 1 (EtherCAT)/+FS1-3K1 (BK1120)/+FS1-3K6 (EL2809)
//     PlcTask Outputs/EAs_0000.a_FR_0300_SEW_Netzschuetz_Versorgungsmodul_EIN_1Min_10sec_Ein_Ausschaltzeit <-> Channel 1/Output
//     PlcTask Outputs/EAs_0000.a_FS1_3K6_Channel_10 <-> Channel 10/Output
//     PlcTask Outputs/EAs_0000.a_FS1_3K6_Channel_11 <-> Channel 11/Output
//     PlcTask Outputs/EAs_0000.a_FS1_3K6_Channel_12 <-> Channel 12/Output
//     PlcTask Outputs/EAs_0000.a_FS1_3K6_Channel_13 <-> Channel 13/Output
//     PlcTask Outputs/EAs_0000.a_FS1_3K6_Channel_14 <-> Channel 14/Output
//     PlcTask Outputs/EAs_0000.a_FS1_3K6_Channel_15 <-> Channel 15/Output
//     PlcTask Outputs/EAs_0000.a_FS1_3K6_Channel_16 <-> Channel 16/Output
//     PlcTask Outputs/EAs_0000.a_FS1_3K6_Channel_2 <-> Channel 2/Output
//     PlcTask Outputs/EAs_0000.a_FS1_3K6_Channel_3 <-> Channel 3/Output
//     PlcTask Outputs/EAs_0000.a_FS1_3K6_Channel_4 <-> Channel 4/Output
//     PlcTask Outputs/EAs_0000.a_FS1_3K6_Channel_5 <-> Channel 5/Output
//     PlcTask Outputs/EAs_0000.a_FS1_3K6_Channel_6 <-> Channel 6/Output
//     PlcTask Outputs/EAs_0000.a_FS1_3K6_Channel_7 <-> Channel 7/Output
//     PlcTask Outputs/EAs_0000.a_FS1_3K6_Channel_8 <-> Channel 8/Output
//     PlcTask Outputs/EAs_0000.a_FS1_3K6_Channel_9 <-> Channel 9/Output
//   (this object) <-> Device 1 (EtherCAT)/+K110-1K1 (BK1120)/+K110-1K2 (EL1809)
//     PlcTask Inputs/EAs_3100.e_FR_3100_Schlossbearbeitung_Bohraggregat_1_Vorlegehub_ist_hinten <-> Channel 2/Input
//     PlcTask Inputs/EAs_3100.e_FR_3100_Schlossbearbeitung_Bohraggregat_3_Vorlegehub_ist_hinten <-> Channel 6/Input
//     PlcTask Inputs/EAs_3100.e_FR_3100_Schlossbearbeitung_Bohraggregat_1_Vorlegehub_ist_vorne <-> Channel 1/Input
//     PlcTask Inputs/EAs_3100.e_FR_3100_Schlossbearbeitung_Bohraggregat_3_Vorlegehub_ist_vorne <-> Channel 5/Input
//     PlcTask Inputs/EAs_3100.e_FR_3100_Schlossbearbeitung_Bohraggregat_2_Bohrhub_ist_hinten <-> Channel 4/Input
//     PlcTask Inputs/EAs_3100.e_FR_3100_Schlossbearbeitung_Bohraggregat_2_Bohrhub_ist_vorne <-> Channel 3/Input
//     PlcTask Inputs/EAs_3200.e_FR_3200_Bandbearbeitung_Bohraggregat_4_Bohrhub_ist_hinten <-> Channel 8/Input
//     PlcTask Inputs/EAs_3200.e_FR_3200_Bandbearbeitung_Bohraggregat_4_Bohrhub_ist_vorne <-> Channel 7/Input
//     PlcTask Inputs/EAs_3200.e_FR_3200_Bandbearbeitung_Bohraggregat_5_Vorlegehub_ist_hinten <-> Channel 10/Input
//     PlcTask Inputs/EAs_3200.e_FR_3200_Bandbearbeitung_Bohraggregat_5_Vorlegehub_ist_vorne <-> Channel 9/Input
//     PlcTask Inputs/EAs_3200.e_FR_3200_Bandbearbeitung_Pusher_ist_hinten <-> Channel 11/Input
//     PlcTask Inputs/EAs_3300.e_FR_3300_Druecker_Schluesselloch_unten_Bohraggregat_6_Bohrhub_ist_oben <-> Channel 12/Input
//     PlcTask Inputs/EAs_3300.e_FR_3300_Druecker_Schluesselloch_unten_Bohraggregat_6_Bohrhub_ist_unten <-> Channel 13/Input
//     PlcTask Inputs/EAs_3400.e_FR_3400_Druecker_Schluesselloch_oben_Bohraggregat_7_Bohrhub_ist_oben <-> Channel 14/Input
//     PlcTask Inputs/EAs_3400.e_FR_3400_Druecker_Schluesselloch_oben_Bohraggregat_7_Bohrhub_ist_unten <-> Channel 15/Input
//     PlcTask Inputs/EAs_3510.e_FR_3510_Transport_Schlossseite_Riemenfoerderer_langsam <-> Channel 16/Input
//   (this object) <-> Device 1 (EtherCAT)/+K110-1K1 (BK1120)/+K110-1K3 (EL1809)
//     PlcTask Inputs/EAs_0000.e_K110_1K3_Channel_10 <-> Channel 10/Input
//     PlcTask Inputs/EAs_0000.e_K110_1K3_Channel_11 <-> Channel 11/Input
//     PlcTask Inputs/EAs_0000.e_K110_1K3_Channel_12 <-> Channel 12/Input
//     PlcTask Inputs/EAs_0000.e_K110_1K3_Channel_13 <-> Channel 13/Input
//     PlcTask Inputs/EAs_0000.e_K110_1K3_Channel_14 <-> Channel 14/Input
//     PlcTask Inputs/EAs_0000.e_K110_1K3_Channel_15 <-> Channel 15/Input
//     PlcTask Inputs/EAs_0000.e_K110_1K3_Channel_16 <-> Channel 16/Input
//     PlcTask Inputs/EAs_3510.e_FR_3510_Transport_Schlossseite_Laengsanschlag_ist_oben <-> Channel 2/Input
//     PlcTask Inputs/EAs_3510.e_FR_3510_Transport_Schlossseite_Laengsanschlag_ist_unten <-> Channel 3/Input
//     PlcTask Inputs/EAs_3510.e_FR_3510_Transport_Schlossseite_Riemenfoerderer_stopp <-> Channel 1/Input
//     PlcTask Inputs/EAs_3520.e_FR_3520_Transport_Bandseite_Laengsanschlag_oben <-> Channel 4/Input
//     PlcTask Inputs/EAs_3520.e_FR_3520_Transport_Bandseite_Laengsanschlag_unten <-> Channel 5/Input
//     PlcTask Inputs/EAs_3540.e_FR_3540_Niederhalter_Bandseite_Niederhalter_Auslauf_ist_oben <-> Channel 8/Input
//     PlcTask Inputs/EAs_3540.e_FR_3540_Niederhalter_Bandseite_Niederhalter_Auslauf_ist_unten <-> Channel 9/Input
//     PlcTask Inputs/EAs_3540.e_FR_3540_Niederhalter_Bandseite_Niederhalter_Einlauf_ist_oben <-> Channel 6/Input
//     PlcTask Inputs/EAs_3540.e_FR_3540_Niederhalter_Bandseite_Niederhalter_Einlauf_ist_unten <-> Channel 7/Input
//   (this object) <-> Device 1 (EtherCAT)/+K110-1K1 (BK1120)/+K110-1K4 (EL1104)
//     PlcTask Inputs/EAs_3100.e_FR_3100_Schlossbearbeitung_Nullkante_Auslauf_ist_oben <-> Channel 3/Input
//     PlcTask Inputs/EAs_3100.e_FR_3100_Schlossbearbeitung_Nullkante_Auslauf_ist_unten <-> Channel 4/Input
//     PlcTask Inputs/EAs_3100.e_FR_3100_Schlossbearbeitung_Nullkante_Einlauf_ist_oben <-> Channel 1/Input
//     PlcTask Inputs/EAs_3100.e_FR_3100_Schlossbearbeitung_Nullkante_Einlauf_ist_unten <-> Channel 2/Input
//   (this object) <-> Device 1 (EtherCAT)/+K110-1K1 (BK1120)/+K110-1K5 (EL1104)
//     PlcTask Inputs/EAs_3510.e_FR_3510_Transport_Schlossseite_X_Achse_Laengsanschlag_Referenz <-> Channel 1/Input
//     PlcTask Inputs/EAs_3520.e_FR_3520_Transport_Bandseite_X_Achse_Laengsanschlag_Referenz <-> Channel 2/Input
//     PlcTask Inputs/EAs_3530.e_FR_3530_Niederhalter_Schlossseite_Niederhalter_Einlauf_ist_oben <-> Channel 3/Input
//     PlcTask Inputs/EAs_3530.e_FR_3530_Niederhalter_Schlossseite_Niederhalter_Einlauf_ist_unten <-> Channel 4/Input
//   (this object) <-> Device 1 (EtherCAT)/+K110-1K1 (BK1120)/+K110-1K6 (EL1104)
//     PlcTask Inputs/EAs_0000.e_K110_1K6_Channel_3 <-> Channel 3/Input
//     PlcTask Inputs/EAs_0000.e_K110_1K6_Channel_4 <-> Channel 4/Input
//     PlcTask Inputs/EAs_3530.e_FR_3530_Niederhalter_Schlossseite_Niederhalter_Auslauf_ist_oben <-> Channel 1/Input
//     PlcTask Inputs/EAs_3530.e_FR_3530_Niederhalter_Schlossseite_Niederhalter_Auslauf_ist_unten <-> Channel 2/Input
//   (this object) <-> Device 1 (EtherCAT)/+K110-1K1 (BK1120)/+K110-2K1 (EL2809)
//     PlcTask Outputs/EAs_3100.a_FR_3100_Schlossbearbeitung_Bohraggregat_1_Vorlegehub_vor <-> Channel 1/Output
//     PlcTask Outputs/EAs_3100.a_FR_3100_Schlossbearbeitung_Bohraggregat_3_Vorlegehub_vor <-> Channel 5/Output
//     PlcTask Outputs/EAs_3100.a_FR_3100_Schlossbearbeitung_Bohraggregat_1_Vorlegehub_zurueck <-> Channel 2/Output
//     PlcTask Outputs/EAs_3100.a_FR_3100_Schlossbearbeitung_Bohraggregat_3_Vorlegehub_zurueck <-> Channel 6/Output
//     PlcTask Outputs/EAs_3100.a_FR_3100_Schlossbearbeitung_Bohraggregat_2_Bohrhub_vor <-> Channel 3/Output
//     PlcTask Outputs/EAs_3100.a_FR_3100_Schlossbearbeitung_Bohraggregat_2_Bohrhub_zurueck <-> Channel 4/Output
//     PlcTask Outputs/EAs_3200.a_FR_3200_Bandbearbeitung_Bohraggregat_4_Bohrhub_vor <-> Channel 7/Output
//     PlcTask Outputs/EAs_3200.a_FR_3200_Bandbearbeitung_Bohraggregat_4_Bohrhub_zurueck <-> Channel 8/Output
//     PlcTask Outputs/EAs_3200.a_FR_3200_Bandbearbeitung_Bohraggregat_5_Vorlegehub_vor <-> Channel 9/Output
//     PlcTask Outputs/EAs_3200.a_FR_3200_Bandbearbeitung_Bohraggregat_5_Vorlegehub_zurueck <-> Channel 10/Output
//     PlcTask Outputs/EAs_3200.a_FR_3200_Bandbearbeitung_Pusher_vor <-> Channel 11/Output
//     PlcTask Outputs/EAs_3200.a_FR_3200_Bandbearbeitung_Pusher_zurueck <-> Channel 12/Output
//     PlcTask Outputs/EAs_3300.a_FR_3300_Druecker_Schluesselloch_unten_Bohraggregat_6_Bohrhub_heben <-> Channel 13/Output
//     PlcTask Outputs/EAs_3300.a_FR_3300_Druecker_Schluesselloch_unten_Bohraggregat_6_Bohrhub_senken <-> Channel 14/Output
//     PlcTask Outputs/EAs_3400.a_FR_3400_Druecker_Schluesselloch_oben_Bohraggregat_7_Bohrhub_heben <-> Channel 15/Output
//     PlcTask Outputs/EAs_3400.a_FR_3400_Druecker_Schluesselloch_oben_Bohraggregat_7_Bohrhub_senken <-> Channel 16/Output
//   (this object) <-> Device 1 (EtherCAT)/+K110-1K1 (BK1120)/+K110-2K2 (EL2809)
//     PlcTask Outputs/EAs_3510.a_FR_3510_Transport_Schlossseite_Laengsanschlag_heben <-> Channel 2/Output
//     PlcTask Outputs/EAs_3510.a_FR_3510_Transport_Schlossseite_Laengsanschlag_senken <-> Channel 3/Output
//     PlcTask Outputs/EAs_3510.a_FR_3510_Transport_Schlossseite_X_Achse_Laengsanschlag_Schienenklemmung_klemmen <-> Channel 1/Output
//     PlcTask Outputs/EAs_3520.a_FR_3520_Transport_Bandseite_Laengsanschlag_Clamp_X_axis_rail_clamp <-> Channel 6/Output
//     PlcTask Outputs/EAs_3520.a_FR_3520_Transport_Bandseite_Laengsanschlag_heben <-> Channel 4/Output
//     PlcTask Outputs/EAs_3520.a_FR_3520_Transport_Bandseite_Laengsanschlag_senken <-> Channel 5/Output
//     PlcTask Outputs/EAs_3540.a_FR_3540_Niederhalter_Bandseite_Niederhalter_heben <-> Channel 7/Output
//     PlcTask Outputs/EAs_3540.a_FR_3540_Niederhalter_Bandseite_Niederhalter_senken <-> Channel 8/Output
//   (this object) <-> Device 1 (EtherCAT)/+K110-1K1 (BK1120)/+K110-2K3 (EL2808)
//     PlcTask Outputs/EAs_3100.a_FR_3100_Schlossbearbeitung_Nullkante_heben <-> Channel 2/Output
//     PlcTask Outputs/EAs_3100.a_FR_3100_Schlossbearbeitung_Nullkante_senken <-> Channel 3/Output
//     PlcTask Outputs/EAs_3100.a_FR_3100_Schlossbearbeitung_Y_Achse_Schienenklemmung_klemmen <-> Channel 1/Output
//     PlcTask Outputs/EAs_3200.a_FR_3200_Bandbearbeitung_Y_Achse_Schienenklemmung_klemmen <-> Channel 4/Output
//     PlcTask Outputs/EAs_3530.a_FR_3530_Niederhalter_Schlossseite_Niederhalter_heben <-> Channel 5/Output
//     PlcTask Outputs/EAs_3530.a_FR_3530_Niederhalter_Schlossseite_Niederhalter_senken <-> Channel 6/Output
//   (this object) <-> Device 1 (EtherCAT)/=3100+FS2-16T1 (Bohraggr Schlosskastenfräser)
//     PlcTask Inputs/EAs_3100.e_Bohraggr_Schlosskast/PD_1_STATUSWORT <-> Module 1 (Standard 16 PD)/Inputs 16 PD/PI 1
//     PlcTask Inputs/EAs_3100.e_Bohraggr_Schlosskast/PD_2_IST_DREHZAHL <-> Module 1 (Standard 16 PD)/Inputs 16 PD/PI 2
//     PlcTask Inputs/EAs_3100.e_Bohraggr_Schlosskast/PD_3_Status <-> Module 1 (Standard 16 PD)/Inputs 16 PD/PI 3
//     PlcTask Inputs/EAs_3100.e_Bohraggr_Schlosskast/PD_4_IST_DREHMOMENT <-> Module 1 (Standard 16 PD)/Inputs 16 PD/PI 4
//     PlcTask Inputs/EAs_3100.e_Bohraggr_Schlosskast/PD_5_IST_STROM <-> Module 1 (Standard 16 PD)/Inputs 16 PD/PI 5
//     PlcTask Outputs/EAs_3100.a_Bohraggr_Schlosskast/PD_1_Steuerwort <-> Module 1 (Standard 16 PD)/Outputs 16 PD/PO 1
//     PlcTask Outputs/EAs_3100.a_Bohraggr_Schlosskast/PD_2_Solldrehzahl <-> Module 1 (Standard 16 PD)/Outputs 16 PD/PO 2
//     PlcTask Outputs/EAs_3100.a_Bohraggr_Schlosskast/PD_3_Sollbeschleunigung <-> Module 1 (Standard 16 PD)/Outputs 16 PD/PO 3
//     PlcTask Outputs/EAs_3100.a_Bohraggr_Schlosskast/PD_4_Sollverzoegerung <-> Module 1 (Standard 16 PD)/Outputs 16 PD/PO 4
//     PlcTask Outputs/EAs_3100.a_Bohraggr_Schlosskast/PD_5_Digitalausgaenge <-> Module 1 (Standard 16 PD)/Outputs 16 PD/PO 5
//   (this object) <-> Device 1 (EtherCAT)/=3100+FS2-17T1 (Bohraggr Vorbohren)
//     PlcTask Inputs/EAs_3100.e_Bohraggr_Vorbohren/PD_1_STATUSWORT <-> Module 1 (Standard 16 PD)/Inputs 16 PD/PI 1
//     PlcTask Inputs/EAs_3100.e_Bohraggr_Vorbohren/PD_2_IST_DREHZAHL <-> Module 1 (Standard 16 PD)/Inputs 16 PD/PI 2
//     PlcTask Inputs/EAs_3100.e_Bohraggr_Vorbohren/PD_3_Status <-> Module 1 (Standard 16 PD)/Inputs 16 PD/PI 3
//     PlcTask Inputs/EAs_3100.e_Bohraggr_Vorbohren/PD_4_IST_DREHMOMENT <-> Module 1 (Standard 16 PD)/Inputs 16 PD/PI 4
//     PlcTask Inputs/EAs_3100.e_Bohraggr_Vorbohren/PD_5_IST_STROM <-> Module 1 (Standard 16 PD)/Inputs 16 PD/PI 5
//     PlcTask Outputs/EAs_3100.a_Bohraggr_Vorbohren/PD_1_Steuerwort <-> Module 1 (Standard 16 PD)/Outputs 16 PD/PO 1
//     PlcTask Outputs/EAs_3100.a_Bohraggr_Vorbohren/PD_2_Solldrehzahl <-> Module 1 (Standard 16 PD)/Outputs 16 PD/PO 2
//     PlcTask Outputs/EAs_3100.a_Bohraggr_Vorbohren/PD_3_Sollbeschleunigung <-> Module 1 (Standard 16 PD)/Outputs 16 PD/PO 3
//     PlcTask Outputs/EAs_3100.a_Bohraggr_Vorbohren/PD_4_Sollverzoegerung <-> Module 1 (Standard 16 PD)/Outputs 16 PD/PO 4
//     PlcTask Outputs/EAs_3100.a_Bohraggr_Vorbohren/PD_5_Digitalausgaenge <-> Module 1 (Standard 16 PD)/Outputs 16 PD/PO 5
//   (this object) <-> Device 1 (EtherCAT)/=3100+FS2-18T1 (Bohraggr Stulpfräser)
//     PlcTask Inputs/EAs_3100.e_Bohraggr_Stulpfraes/PD_1_STATUSWORT <-> Module 1 (Standard 16 PD)/Inputs 16 PD/PI 1
//     PlcTask Inputs/EAs_3100.e_Bohraggr_Stulpfraes/PD_2_IST_DREHZAHL <-> Module 1 (Standard 16 PD)/Inputs 16 PD/PI 2
//     PlcTask Inputs/EAs_3100.e_Bohraggr_Stulpfraes/PD_3_Status <-> Module 1 (Standard 16 PD)/Inputs 16 PD/PI 3
//     PlcTask Inputs/EAs_3100.e_Bohraggr_Stulpfraes/PD_4_IST_DREHMOMENT <-> Module 1 (Standard 16 PD)/Inputs 16 PD/PI 4
//     PlcTask Inputs/EAs_3100.e_Bohraggr_Stulpfraes/PD_5_IST_STROM <-> Module 1 (Standard 16 PD)/Inputs 16 PD/PI 5
//     PlcTask Outputs/EAs_3100.a_Bohraggr_Stulpfraes/PD_1_Steuerwort <-> Module 1 (Standard 16 PD)/Outputs 16 PD/PO 1
//     PlcTask Outputs/EAs_3100.a_Bohraggr_Stulpfraes/PD_2_Solldrehzahl <-> Module 1 (Standard 16 PD)/Outputs 16 PD/PO 2
//     PlcTask Outputs/EAs_3100.a_Bohraggr_Stulpfraes/PD_3_Sollbeschleunigung <-> Module 1 (Standard 16 PD)/Outputs 16 PD/PO 3
//     PlcTask Outputs/EAs_3100.a_Bohraggr_Stulpfraes/PD_4_Sollverzoegerung <-> Module 1 (Standard 16 PD)/Outputs 16 PD/PO 4
//     PlcTask Outputs/EAs_3100.a_Bohraggr_Stulpfraes/PD_5_Digitalausgaenge <-> Module 1 (Standard 16 PD)/Outputs 16 PD/PO 5
//   (this object) <-> Device 1 (EtherCAT)/=3200+FS2-16T1 (Bohraggr Stufenbohrer)
//     PlcTask Inputs/EAs_3200.e_Bohraggr_Stufenbohr/PD_1_STATUSWORT <-> Module 1 (Standard 16 PD)/Inputs 16 PD/PI 1
//     PlcTask Inputs/EAs_3200.e_Bohraggr_Stufenbohr/PD_2_IST_DREHZAHL <-> Module 1 (Standard 16 PD)/Inputs 16 PD/PI 2
//     PlcTask Inputs/EAs_3200.e_Bohraggr_Stufenbohr/PD_3_Status <-> Module 1 (Standard 16 PD)/Inputs 16 PD/PI 3
//     PlcTask Inputs/EAs_3200.e_Bohraggr_Stufenbohr/PD_4_IST_DREHMOMENT <-> Module 1 (Standard 16 PD)/Inputs 16 PD/PI 4
//     PlcTask Inputs/EAs_3200.e_Bohraggr_Stufenbohr/PD_5_IST_STROM <-> Module 1 (Standard 16 PD)/Inputs 16 PD/PI 5
//     PlcTask Outputs/EAs_3200.a_Bohraggr_Stufenbohr/PD_1_Steuerwort <-> Module 1 (Standard 16 PD)/Outputs 16 PD/PO 1
//     PlcTask Outputs/EAs_3200.a_Bohraggr_Stufenbohr/PD_2_Solldrehzahl <-> Module 1 (Standard 16 PD)/Outputs 16 PD/PO 2
//     PlcTask Outputs/EAs_3200.a_Bohraggr_Stufenbohr/PD_3_Sollbeschleunigung <-> Module 1 (Standard 16 PD)/Outputs 16 PD/PO 3
//     PlcTask Outputs/EAs_3200.a_Bohraggr_Stufenbohr/PD_4_Sollverzoegerung <-> Module 1 (Standard 16 PD)/Outputs 16 PD/PO 4
//     PlcTask Outputs/EAs_3200.a_Bohraggr_Stufenbohr/PD_5_Digitalausgaenge <-> Module 1 (Standard 16 PD)/Outputs 16 PD/PO 5
//   (this object) <-> Device 1 (EtherCAT)/=3200+FS2-17T1 (Bohraggr Stulpfräser)
//     PlcTask Inputs/EAs_3200.e_Bohraggr_Stulpfraes/PD_1_STATUSWORT <-> Module 1 (Standard 16 PD)/Inputs 16 PD/PI 1
//     PlcTask Inputs/EAs_3200.e_Bohraggr_Stulpfraes/PD_2_IST_DREHZAHL <-> Module 1 (Standard 16 PD)/Inputs 16 PD/PI 2
//     PlcTask Inputs/EAs_3200.e_Bohraggr_Stulpfraes/PD_3_Status <-> Module 1 (Standard 16 PD)/Inputs 16 PD/PI 3
//     PlcTask Inputs/EAs_3200.e_Bohraggr_Stulpfraes/PD_4_IST_DREHMOMENT <-> Module 1 (Standard 16 PD)/Inputs 16 PD/PI 4
//     PlcTask Inputs/EAs_3200.e_Bohraggr_Stulpfraes/PD_5_IST_STROM <-> Module 1 (Standard 16 PD)/Inputs 16 PD/PI 5
//     PlcTask Outputs/EAs_3200.a_Bohraggr_Stulpfraes/PD_1_Steuerwort <-> Module 1 (Standard 16 PD)/Outputs 16 PD/PO 1
//     PlcTask Outputs/EAs_3200.a_Bohraggr_Stulpfraes/PD_2_Solldrehzahl <-> Module 1 (Standard 16 PD)/Outputs 16 PD/PO 2
//     PlcTask Outputs/EAs_3200.a_Bohraggr_Stulpfraes/PD_3_Sollbeschleunigung <-> Module 1 (Standard 16 PD)/Outputs 16 PD/PO 3
//     PlcTask Outputs/EAs_3200.a_Bohraggr_Stulpfraes/PD_4_Sollverzoegerung <-> Module 1 (Standard 16 PD)/Outputs 16 PD/PO 4
//     PlcTask Outputs/EAs_3200.a_Bohraggr_Stulpfraes/PD_5_Digitalausgaenge <-> Module 1 (Standard 16 PD)/Outputs 16 PD/PO 5
//   (this object) <-> Device 1 (EtherCAT)/=3300+FS2-16T1 (Bohraggr Schlüsselloch unten)
//     PlcTask Inputs/EAs_3300.e_Bohraggr_Schluessel_un/PD_1_STATUSWORT <-> Module 1 (Standard 16 PD)/Inputs 16 PD/PI 1
//     PlcTask Inputs/EAs_3300.e_Bohraggr_Schluessel_un/PD_2_IST_DREHZAHL <-> Module 1 (Standard 16 PD)/Inputs 16 PD/PI 2
//     PlcTask Inputs/EAs_3300.e_Bohraggr_Schluessel_un/PD_3_Status <-> Module 1 (Standard 16 PD)/Inputs 16 PD/PI 3
//     PlcTask Inputs/EAs_3300.e_Bohraggr_Schluessel_un/PD_4_IST_DREHMOMENT <-> Module 1 (Standard 16 PD)/Inputs 16 PD/PI 4
//     PlcTask Inputs/EAs_3300.e_Bohraggr_Schluessel_un/PD_5_IST_STROM <-> Module 1 (Standard 16 PD)/Inputs 16 PD/PI 5
//     PlcTask Outputs/EAs_3300.a_Bohraggr_Schluessel_un/PD_1_Steuerwort <-> Module 1 (Standard 16 PD)/Outputs 16 PD/PO 1
//     PlcTask Outputs/EAs_3300.a_Bohraggr_Schluessel_un/PD_2_Solldrehzahl <-> Module 1 (Standard 16 PD)/Outputs 16 PD/PO 2
//     PlcTask Outputs/EAs_3300.a_Bohraggr_Schluessel_un/PD_3_Sollbeschleunigung <-> Module 1 (Standard 16 PD)/Outputs 16 PD/PO 3
//     PlcTask Outputs/EAs_3300.a_Bohraggr_Schluessel_un/PD_4_Sollverzoegerung <-> Module 1 (Standard 16 PD)/Outputs 16 PD/PO 4
//     PlcTask Outputs/EAs_3300.a_Bohraggr_Schluessel_un/PD_5_Digitalausgaenge <-> Module 1 (Standard 16 PD)/Outputs 16 PD/PO 5
//   (this object) <-> Device 1 (EtherCAT)/=3400+FS2-16T1 (Bohraggr Schlüsselloch oben)
//     PlcTask Inputs/EAs_3400.e_Bohraggr_Schluessel_ob/PD_1_STATUSWORT <-> Module 1 (Standard 16 PD)/Inputs 16 PD/PI 1
//     PlcTask Inputs/EAs_3400.e_Bohraggr_Schluessel_ob/PD_2_IST_DREHZAHL <-> Module 1 (Standard 16 PD)/Inputs 16 PD/PI 2
//     PlcTask Inputs/EAs_3400.e_Bohraggr_Schluessel_ob/PD_3_Status <-> Module 1 (Standard 16 PD)/Inputs 16 PD/PI 3
//     PlcTask Inputs/EAs_3400.e_Bohraggr_Schluessel_ob/PD_4_IST_DREHMOMENT <-> Module 1 (Standard 16 PD)/Inputs 16 PD/PI 4
//     PlcTask Inputs/EAs_3400.e_Bohraggr_Schluessel_ob/PD_5_IST_STROM <-> Module 1 (Standard 16 PD)/Inputs 16 PD/PI 5
//     PlcTask Outputs/EAs_3400.a_Bohraggr_Schluessel_ob/PD_1_Steuerwort <-> Module 1 (Standard 16 PD)/Outputs 16 PD/PO 1
//     PlcTask Outputs/EAs_3400.a_Bohraggr_Schluessel_ob/PD_2_Solldrehzahl <-> Module 1 (Standard 16 PD)/Outputs 16 PD/PO 2
//     PlcTask Outputs/EAs_3400.a_Bohraggr_Schluessel_ob/PD_3_Sollbeschleunigung <-> Module 1 (Standard 16 PD)/Outputs 16 PD/PO 3
//     PlcTask Outputs/EAs_3400.a_Bohraggr_Schluessel_ob/PD_4_Sollverzoegerung <-> Module 1 (Standard 16 PD)/Outputs 16 PD/PO 4
//     PlcTask Outputs/EAs_3400.a_Bohraggr_Schluessel_ob/PD_5_Digitalausgaenge <-> Module 1 (Standard 16 PD)/Outputs 16 PD/PO 5
//   (this object) <-> Device 1 (EtherCAT)/=3510+FS2-6T1 (Transport Schlossseite X-Achse)
//     PlcTask Inputs/EAs_3510.e_Trans_Schlossseite/PD_1_STATUSWORT <-> Module 1 (Standard 16 PD)/Inputs 16 PD/PI 1
//     PlcTask Inputs/EAs_3510.e_Trans_Schlossseite/PD_2_IST_DREHZAHL <-> Module 1 (Standard 16 PD)/Inputs 16 PD/PI 2
//     PlcTask Inputs/EAs_3510.e_Trans_Schlossseite/PD_3_Status <-> Module 1 (Standard 16 PD)/Inputs 16 PD/PI 3
//     PlcTask Inputs/EAs_3510.e_Trans_Schlossseite/PD_4_IST_DREHMOMENT <-> Module 1 (Standard 16 PD)/Inputs 16 PD/PI 4
//     PlcTask Inputs/EAs_3510.e_Trans_Schlossseite/PD_5_IST_STROM <-> Module 1 (Standard 16 PD)/Inputs 16 PD/PI 5
//     PlcTask Outputs/EAs_3510.a_Trans_Schlossseite/PD_1_Steuerwort <-> Module 1 (Standard 16 PD)/Outputs 16 PD/PO 1
//     PlcTask Outputs/EAs_3510.a_Trans_Schlossseite/PD_2_Solldrehzahl <-> Module 1 (Standard 16 PD)/Outputs 16 PD/PO 2
//     PlcTask Outputs/EAs_3510.a_Trans_Schlossseite/PD_3_Sollbeschleunigung <-> Module 1 (Standard 16 PD)/Outputs 16 PD/PO 3
//     PlcTask Outputs/EAs_3510.a_Trans_Schlossseite/PD_4_Sollverzoegerung <-> Module 1 (Standard 16 PD)/Outputs 16 PD/PO 4
//     PlcTask Outputs/EAs_3510.a_Trans_Schlossseite/PD_5_Digitalausgaenge <-> Module 1 (Standard 16 PD)/Outputs 16 PD/PO 5
//   (this object) <-> Device 1 (EtherCAT)/=3520+FS2-6T1 (Transport Bandseite X-Achse)
//     PlcTask Inputs/EAs_3520.e_Trans_Bandseite/PD_1_STATUSWORT <-> Module 1 (Standard 16 PD)/Inputs 16 PD/PI 1
//     PlcTask Inputs/EAs_3520.e_Trans_Bandseite/PD_2_IST_DREHZAHL <-> Module 1 (Standard 16 PD)/Inputs 16 PD/PI 2
//     PlcTask Inputs/EAs_3520.e_Trans_Bandseite/PD_3_Status <-> Module 1 (Standard 16 PD)/Inputs 16 PD/PI 3
//     PlcTask Inputs/EAs_3520.e_Trans_Bandseite/PD_4_IST_DREHMOMENT <-> Module 1 (Standard 16 PD)/Inputs 16 PD/PI 4
//     PlcTask Inputs/EAs_3520.e_Trans_Bandseite/PD_5_IST_STROM <-> Module 1 (Standard 16 PD)/Inputs 16 PD/PI 5
//     PlcTask Outputs/EAs_3520.a_Trans_Bandseite/PD_1_Steuerwort <-> Module 1 (Standard 16 PD)/Outputs 16 PD/PO 1
//     PlcTask Outputs/EAs_3520.a_Trans_Bandseite/PD_2_Solldrehzahl <-> Module 1 (Standard 16 PD)/Outputs 16 PD/PO 2
//     PlcTask Outputs/EAs_3520.a_Trans_Bandseite/PD_3_Sollbeschleunigung <-> Module 1 (Standard 16 PD)/Outputs 16 PD/PO 3
//     PlcTask Outputs/EAs_3520.a_Trans_Bandseite/PD_4_Sollverzoegerung <-> Module 1 (Standard 16 PD)/Outputs 16 PD/PO 4
//     PlcTask Outputs/EAs_3520.a_Trans_Bandseite/PD_5_Digitalausgaenge <-> Module 1 (Standard 16 PD)/Outputs 16 PD/PO 5
//   (this object) <-> NC-Task 1 SAF/Axes/=3100+FS2-11M1 (X-Achse)
//     PlcTask Inputs/EAs_3100.ea_X_Achse.NcToPlc <-> Outputs/ToPlc
//     PlcTask Outputs/EAs_3100.ea_X_Achse.PlcToNc <-> Inputs/FromPlc
//   (this object) <-> NC-Task 1 SAF/Axes/=3100+FS2-12M1 (Y-Achse)
//     PlcTask Inputs/EAs_3100.ea_Y_Achse.NcToPlc <-> Outputs/ToPlc
//     PlcTask Outputs/EAs_3100.ea_Y_Achse.PlcToNc <-> Inputs/FromPlc
//   (this object) <-> NC-Task 1 SAF/Axes/=3100+FS2-13M1 (Z-Achse)
//     PlcTask Inputs/EAs_3100.ea_Z_Achse.NcToPlc <-> Outputs/ToPlc
//     PlcTask Outputs/EAs_3100.ea_Z_Achse.PlcToNc <-> Inputs/FromPlc
//   (this object) <-> NC-Task 1 SAF/Axes/=3200+FS2-11M1 (X-Achse)
//     PlcTask Inputs/EAs_3200.ea_X_Achse.NcToPlc <-> Outputs/ToPlc
//     PlcTask Outputs/EAs_3200.ea_X_Achse.PlcToNc <-> Inputs/FromPlc
//   (this object) <-> NC-Task 1 SAF/Axes/=3200+FS2-12M1 (Y-Achse)
//     PlcTask Inputs/EAs_3200.ea_Y_Achse.NcToPlc <-> Outputs/ToPlc
//     PlcTask Outputs/EAs_3200.ea_Y_Achse.PlcToNc <-> Inputs/FromPlc
//   (this object) <-> NC-Task 1 SAF/Axes/=3200+FS2-13M1 (Z-Achse)
//     PlcTask Inputs/EAs_3200.ea_Z_Achse.NcToPlc <-> Outputs/ToPlc
//     PlcTask Outputs/EAs_3200.ea_Z_Achse.PlcToNc <-> Inputs/FromPlc
//   (this object) <-> NC-Task 1 SAF/Axes/=3300+FS2-11M1 (X-Achse)
//     PlcTask Inputs/EAs_3300.ea_X_Achse.NcToPlc <-> Outputs/ToPlc
//     PlcTask Outputs/EAs_3300.ea_X_Achse.PlcToNc <-> Inputs/FromPlc
//   (this object) <-> NC-Task 1 SAF/Axes/=3300+FS2-12M1 (Y-Achse)
//     PlcTask Inputs/EAs_3300.ea_Y_Achse.NcToPlc <-> Outputs/ToPlc
//     PlcTask Outputs/EAs_3300.ea_Y_Achse.PlcToNc <-> Inputs/FromPlc
//   (this object) <-> NC-Task 1 SAF/Axes/=3400+FS2-11M1 (X-Achse)
//     PlcTask Inputs/EAs_3400.ea_X_Achse.NcToPlc <-> Outputs/ToPlc
//     PlcTask Outputs/EAs_3400.ea_X_Achse.PlcToNc <-> Inputs/FromPlc
//   (this object) <-> NC-Task 1 SAF/Axes/=3400+FS2-12M1 (Y-Achse)
//     PlcTask Inputs/EAs_3400.ea_Y_Achse.NcToPlc <-> Outputs/ToPlc
//     PlcTask Outputs/EAs_3400.ea_Y_Achse.PlcToNc <-> Inputs/FromPlc
//   (this object) <-> NC-Task 1 SAF/Axes/=3520+FS2-11M1 (Y-Achse)
//     PlcTask Inputs/EAs_3520.ea_Y_Achse.NcToPlc <-> Outputs/ToPlc
//     PlcTask Outputs/EAs_3520.ea_Y_Achse.PlcToNc <-> Inputs/FromPlc
//   (this object) <-> NC-Task 1 SAF/Axes/=3540+FS2-11M1 (Y-Achse)
//     PlcTask Inputs/EAs_3540.ea_Y_Achse.NcToPlc <-> Outputs/ToPlc
//     PlcTask Outputs/EAs_3540.ea_Y_Achse.PlcToNc <-> Inputs/FromPlc

// ---- SRT_Allgemein/0010_Bausteine_mitDuts/DUTs/DUT_Visu_SteuerStatus.TcDUT
TYPE DUT_Visu_SteuerStatus :
STRUCT
	
	hand			: BOOL ;	(*	Handbetrieb anwählen 	*)
	auto			: BOOL ;	(*	Automatik anwählen		*)
	auto_start		: BOOL ;	(*	Automatik Start			*)
	auto_stop		: BOOL ;	(*	Automatik Stop			*)
	auto_pause		: BOOL ;	(*	Automatik Pause			*)
	reset			: BOOL ;	(*	Anlagenreset			*)
	grundstellung	: BOOL ;	(*	Grundstellung anfahren	*)
	einlauf_sperre	: BOOL ;
	auslauf_sperre	: BOOL ;

	auto_aktiv		: BOOL ;	(*	Status an die Visu - Maschinenoverride		*)
	res10			: BOOL ;	(*	*)
	res11			: BOOL ;	(*	*)
	res12			: BOOL ;	(*	*)
	res13			: BOOL ;	(*	*)
	res14			: BOOL ;	(*	*)
	res15			: BOOL ;	(*	*)
	res16			: BOOL ;	(*	*)

END_STRUCT	
END_TYPE

// ---- SRT_Allgemein/0010_Bausteine_mitDuts/DUTs/Meldungen/DUT_Diagnose_3000.TcDUT
TYPE DUT_Diagnose_3000 :
STRUCT
	Nr_001		:DINT;     
	Nr_002		:DINT;
	Nr_003		:DINT;
	Nr_004		:DINT;
	Nr_005		:DINT;
	Nr_006		:DINT;
	Nr_007		:DINT;
	Nr_008		:DINT;
	Nr_009		:DINT;
	Nr_010		:DINT;
	Nr_011		:DINT;
	Nr_012		:DINT;
	Nr_013		:DINT;
	Nr_014		:DINT;
	Nr_015		:DINT;
	Nr_016		:DINT;
	Nr_017		:DINT;
	Nr_018		:DINT;
	Nr_019		:DINT;
	Nr_020		:DINT;
	Nr_021		:DINT;
	Nr_022		:DINT;
	Nr_023		:DINT;
	Nr_024		:DINT;
	Nr_025		:DINT;
	Nr_026		:DINT;
	Nr_027		:DINT;
	Nr_028		:DINT;
	Nr_029		:DINT;
	Nr_030		:DINT;
	Nr_031		:DINT;
	Nr_032		:DINT;
	Nr_033		:DINT;
	Nr_034		:DINT;
	Nr_035		:DINT;
	Nr_036		:DINT;
	Nr_037		:DINT;
	Nr_038		:DINT;
	Nr_039		:DINT;
	Nr_040		:DINT;
	Nr_041		:DINT;
	Nr_042		:DINT;
	Nr_043		:DINT;
	Nr_044		:DINT;
	Nr_045		:DINT;
	Nr_046		:DINT;
	Nr_047		:DINT;
	Nr_048		:DINT;
	Nr_049		:DINT;
	Nr_050		:DINT;
	Nr_051		:DINT;
	Nr_052		:DINT;
	Nr_053		:DINT;
	Nr_054		:DINT;
	Nr_055		:DINT;
	Nr_056		:DINT;
	Nr_057		:DINT;
	Nr_058		:DINT;
	Nr_059		:DINT;
	Nr_060		:DINT;
	Nr_061		:DINT;
	Nr_062		:DINT;
	Nr_063		:DINT;
	Nr_064		:DINT;
	Nr_065		:DINT;
	Nr_066		:DINT;
	Nr_067		:DINT;
	Nr_068		:DINT;
	Nr_069		:DINT;
	Nr_070		:DINT;
	Nr_071		:DINT;
	Nr_072		:DINT;
	Nr_073		:DINT;
	Nr_074		:DINT;
	Nr_075		:DINT;
	Nr_076		:DINT;
	Nr_077		:DINT;
	Nr_078		:DINT;
	Nr_079		:DINT;
	Nr_080		:DINT;
	Nr_081		:DINT;
	Nr_082		:DINT;
	Nr_083		:DINT;
	Nr_084		:DINT;
	Nr_085		:DINT;
	Nr_086		:DINT;
	Nr_087		:DINT;
	Nr_088		:DINT;
	Nr_089		:DINT;
	Nr_090		:DINT;
	Nr_091		:DINT;
	Nr_092		:DINT;
	Nr_093		:DINT;
	Nr_094		:DINT;
	Nr_095		:DINT;
	Nr_096		:DINT;
	Nr_097		:DINT;
	Nr_098		:DINT;
	Nr_099		:DINT;
	Nr_100		:DINT;
	Nr_101		:DINT;
	Nr_102		:DINT;
	Nr_103		:DINT;
	Nr_104		:DINT;
	Nr_105		:DINT;
	Nr_106		:DINT;
	Nr_107		:DINT;
	Nr_108		:DINT;
	Nr_109		:DINT;
	Nr_110		:DINT;
	Nr_111		:DINT;
	Nr_112		:DINT;
	Nr_113		:DINT;
	Nr_114		:DINT;
	Nr_115		:DINT;
	Nr_116		:DINT;
	Nr_117		:DINT;
	Nr_118		:DINT;
	Nr_119		:DINT;
	Nr_120		:DINT;
	Nr_121		:DINT;
	Nr_122		:DINT;
	Nr_123		:DINT;
	Nr_124		:DINT;
	Nr_125		:DINT;
	Nr_126		:DINT;
	Nr_127		:DINT;
	Nr_128		:DINT;
	Nr_129		:DINT;
	Nr_130		:DINT;
	Nr_131		:DINT;
	Nr_132		:DINT;
	Nr_133		:DINT;
	Nr_134		:DINT;
	Nr_135		:DINT;
	Nr_136		:DINT;
	Nr_137		:DINT;
	Nr_138		:DINT;
	Nr_139		:DINT;
	Nr_140		:DINT;
	Nr_141		:DINT;
	Nr_142		:DINT;
	Nr_143		:DINT;
	Nr_144		:DINT;
	Nr_145		:DINT;
	Nr_146		:DINT;
	Nr_147		:DINT;
	Nr_148		:DINT;
	Nr_149		:DINT;
	Nr_150		:DINT;
	Nr_151		:DINT;
	Nr_152		:DINT;
	Nr_153		:DINT;
	Nr_154		:DINT;
	Nr_155		:DINT;
	Nr_156		:DINT;
	Nr_157		:DINT;
	Nr_158		:DINT;
	Nr_159		:DINT;
	Nr_160		:DINT;
	Nr_161		:DINT;
	Nr_162		:DINT;
	Nr_163		:DINT;
	Nr_164		:DINT;
	Nr_165		:DINT;
	Nr_166		:DINT;
	Nr_167		:DINT;
	Nr_168		:DINT;
	Nr_169		:DINT;
	Nr_170		:DINT;
	Nr_171		:DINT;
	Nr_172		:DINT;
	Nr_173		:DINT;
	Nr_174		:DINT;
	Nr_175		:DINT;
	Nr_176		:DINT;
	Nr_177		:DINT;
	Nr_178		:DINT;
	Nr_179		:DINT;
	Nr_180		:DINT;
	Nr_181		:DINT;
	Nr_182		:DINT;
	Nr_183		:DINT;
	Nr_184		:DINT;
	Nr_185		:DINT;
	Nr_186		:DINT;
	Nr_187		:DINT;
	Nr_188		:DINT;
	Nr_189		:DINT;
	Nr_190		:DINT;
	Nr_191		:DINT;
	Nr_192		:DINT;
	Nr_193		:DINT;
	Nr_194		:DINT;
	Nr_195		:DINT;
	Nr_196		:DINT;
	Nr_197		:DINT;
	Nr_198		:DINT;
	Nr_199		:DINT;
	
END_STRUCT
END_TYPE

// ---- SRT_Allgemein/0010_Bausteine_mitDuts/DUTs/Meldungen/DUT_Diagnose_4000.TcDUT
TYPE DUT_Diagnose_4000 :
STRUCT
	Nr_001		:DINT;     
	Nr_002		:DINT;
	Nr_003		:DINT;
	Nr_004		:DINT;
	Nr_005		:DINT;
	Nr_006		:DINT;
	Nr_007		:DINT;
	Nr_008		:DINT;
	Nr_009		:DINT;
	Nr_010		:DINT;
	Nr_011		:DINT;
	Nr_012		:DINT;
	Nr_013		:DINT;
	Nr_014		:DINT;
	Nr_015		:DINT;
	Nr_016		:DINT;
	Nr_017		:DINT;
	Nr_018		:DINT;
	Nr_019		:DINT;
	Nr_020		:DINT;
	Nr_021		:DINT;
	Nr_022		:DINT;
	Nr_023		:DINT;
	Nr_024		:DINT;
	Nr_025		:DINT;
	Nr_026		:DINT;
	Nr_027		:DINT;
	Nr_028		:DINT;
	Nr_029		:DINT;
	Nr_030		:DINT;
	Nr_031		:DINT;
	Nr_032		:DINT;
	Nr_033		:DINT;
	Nr_034		:DINT;
	Nr_035		:DINT;
	Nr_036		:DINT;
	Nr_037		:DINT;
	Nr_038		:DINT;
	Nr_039		:DINT;
	Nr_040		:DINT;
	Nr_041		:DINT;
	Nr_042		:DINT;
	Nr_043		:DINT;
	Nr_044		:DINT;
	Nr_045		:DINT;
	Nr_046		:DINT;
	Nr_047		:DINT;
	Nr_048		:DINT;
	Nr_049		:DINT;
	Nr_050		:DINT;
	Nr_051		:DINT;
	Nr_052		:DINT;
	Nr_053		:DINT;
	Nr_054		:DINT;
	Nr_055		:DINT;
	Nr_056		:DINT;
	Nr_057		:DINT;
	Nr_058		:DINT;
	Nr_059		:DINT;
	Nr_060		:DINT;
	Nr_061		:DINT;
	Nr_062		:DINT;
	Nr_063		:DINT;
	Nr_064		:DINT;
	Nr_065		:DINT;
	Nr_066		:DINT;
	Nr_067		:DINT;
	Nr_068		:DINT;
	Nr_069		:DINT;
	Nr_070		:DINT;
	Nr_071		:DINT;
	Nr_072		:DINT;
	Nr_073		:DINT;
	Nr_074		:DINT;
	Nr_075		:DINT;
	Nr_076		:DINT;
	Nr_077		:DINT;
	Nr_078		:DINT;
	Nr_079		:DINT;
	Nr_080		:DINT;
	Nr_081		:DINT;
	Nr_082		:DINT;
	Nr_083		:DINT;
	Nr_084		:DINT;
	Nr_085		:DINT;
	Nr_086		:DINT;
	Nr_087		:DINT;
	Nr_088		:DINT;
	Nr_089		:DINT;
	Nr_090		:DINT;
	Nr_091		:DINT;
	Nr_092		:DINT;
	Nr_093		:DINT;
	Nr_094		:DINT;
	Nr_095		:DINT;
	Nr_096		:DINT;
	Nr_097		:DINT;
	Nr_098		:DINT;
	Nr_099		:DINT;
	Nr_100		:DINT;
	Nr_101		:DINT;
	Nr_102		:DINT;
	Nr_103		:DINT;
	Nr_104		:DINT;
	Nr_105		:DINT;
	Nr_106		:DINT;
	Nr_107		:DINT;
	Nr_108		:DINT;
	Nr_109		:DINT;
	Nr_110		:DINT;
	Nr_111		:DINT;
	Nr_112		:DINT;
	Nr_113		:DINT;
	Nr_114		:DINT;
	Nr_115		:DINT;
	Nr_116		:DINT;
	Nr_117		:DINT;
	Nr_118		:DINT;
	Nr_119		:DINT;
	Nr_120		:DINT;
	Nr_121		:DINT;
	Nr_122		:DINT;
	Nr_123		:DINT;
	Nr_124		:DINT;
	Nr_125		:DINT;
	Nr_126		:DINT;
	Nr_127		:DINT;
	Nr_128		:DINT;
	Nr_129		:DINT;
	Nr_130		:DINT;
	Nr_131		:DINT;
	Nr_132		:DINT;
	Nr_133		:DINT;
	Nr_134		:DINT;
	Nr_135		:DINT;
	Nr_136		:DINT;
	Nr_137		:DINT;
	Nr_138		:DINT;
	Nr_139		:DINT;
	Nr_140		:DINT;
	Nr_141		:DINT;
	Nr_142		:DINT;
	Nr_143		:DINT;
	Nr_144		:DINT;
	Nr_145		:DINT;
	Nr_146		:DINT;
	Nr_147		:DINT;
	Nr_148		:DINT;
	Nr_149		:DINT;
	Nr_150		:DINT;
	Nr_151		:DINT;
	Nr_152		:DINT;
	Nr_153		:DINT;
	Nr_154		:DINT;
	Nr_155		:DINT;
	Nr_156		:DINT;
	Nr_157		:DINT;
	Nr_158		:DINT;
	Nr_159		:DINT;
	Nr_160		:DINT;
	Nr_161		:DINT;
	Nr_162		:DINT;
	Nr_163		:DINT;
	Nr_164		:DINT;
	Nr_165		:DINT;
	Nr_166		:DINT;
	Nr_167		:DINT;
	Nr_168		:DINT;
	Nr_169		:DINT;
	Nr_170		:DINT;
	Nr_171		:DINT;
	Nr_172		:DINT;
	Nr_173		:DINT;
	Nr_174		:DINT;
	Nr_175		:DINT;
	Nr_176		:DINT;
	Nr_177		:DINT;
	Nr_178		:DINT;
	Nr_179		:DINT;
	Nr_180		:DINT;
	Nr_181		:DINT;
	Nr_182		:DINT;
	Nr_183		:DINT;
	Nr_184		:DINT;
	Nr_185		:DINT;
	Nr_186		:DINT;
	Nr_187		:DINT;
	Nr_188		:DINT;
	Nr_189		:DINT;
	Nr_190		:DINT;
	Nr_191		:DINT;
	Nr_192		:DINT;
	Nr_193		:DINT;
	Nr_194		:DINT;
	Nr_195		:DINT;
	Nr_196		:DINT;
	Nr_197		:DINT;
	Nr_198		:DINT;
	Nr_199		:DINT;
	
END_STRUCT
END_TYPE

// ---- SRT_Allgemein/0010_Bausteine_mitDuts/DUTs/Meldungen/DUT_Diagnose_5000.TcDUT
TYPE DUT_Diagnose_5000 :
STRUCT
	Nr_001		:DINT;     
	Nr_002		:DINT;
	Nr_003		:DINT;
	Nr_004		:DINT;
	Nr_005		:DINT;
	Nr_006		:DINT;
	Nr_007		:DINT;
	Nr_008		:DINT;
	Nr_009		:DINT;
	Nr_010		:DINT;
	Nr_011		:DINT;
	Nr_012		:DINT;
	Nr_013		:DINT;
	Nr_014		:DINT;
	Nr_015		:DINT;
	Nr_016		:DINT;
	Nr_017		:DINT;
	Nr_018		:DINT;
	Nr_019		:DINT;
	Nr_020		:DINT;
	Nr_021		:DINT;
	Nr_022		:DINT;
	Nr_023		:DINT;
	Nr_024		:DINT;
	Nr_025		:DINT;
	Nr_026		:DINT;
	Nr_027		:DINT;
	Nr_028		:DINT;
	Nr_029		:DINT;
	Nr_030		:DINT;
	Nr_031		:DINT;
	Nr_032		:DINT;
	Nr_033		:DINT;
	Nr_034		:DINT;
	Nr_035		:DINT;
	Nr_036		:DINT;
	Nr_037		:DINT;
	Nr_038		:DINT;
	Nr_039		:DINT;
	Nr_040		:DINT;
	Nr_041		:DINT;
	Nr_042		:DINT;
	Nr_043		:DINT;
	Nr_044		:DINT;
	Nr_045		:DINT;
	Nr_046		:DINT;
	Nr_047		:DINT;
	Nr_048		:DINT;
	Nr_049		:DINT;
	Nr_050		:DINT;
	Nr_051		:DINT;
	Nr_052		:DINT;
	Nr_053		:DINT;
	Nr_054		:DINT;
	Nr_055		:DINT;
	Nr_056		:DINT;
	Nr_057		:DINT;
	Nr_058		:DINT;
	Nr_059		:DINT;
	Nr_060		:DINT;
	Nr_061		:DINT;
	Nr_062		:DINT;
	Nr_063		:DINT;
	Nr_064		:DINT;
	Nr_065		:DINT;
	Nr_066		:DINT;
	Nr_067		:DINT;
	Nr_068		:DINT;
	Nr_069		:DINT;
	Nr_070		:DINT;
	Nr_071		:DINT;
	Nr_072		:DINT;
	Nr_073		:DINT;
	Nr_074		:DINT;
	Nr_075		:DINT;
	Nr_076		:DINT;
	Nr_077		:DINT;
	Nr_078		:DINT;
	Nr_079		:DINT;
	Nr_080		:DINT;
	Nr_081		:DINT;
	Nr_082		:DINT;
	Nr_083		:DINT;
	Nr_084		:DINT;
	Nr_085		:DINT;
	Nr_086		:DINT;
	Nr_087		:DINT;
	Nr_088		:DINT;
	Nr_089		:DINT;
	Nr_090		:DINT;
	Nr_091		:DINT;
	Nr_092		:DINT;
	Nr_093		:DINT;
	Nr_094		:DINT;
	Nr_095		:DINT;
	Nr_096		:DINT;
	Nr_097		:DINT;
	Nr_098		:DINT;
	Nr_099		:DINT;
	Nr_100		:DINT;
	Nr_101		:DINT;
	Nr_102		:DINT;
	Nr_103		:DINT;
	Nr_104		:DINT;
	Nr_105		:DINT;
	Nr_106		:DINT;
	Nr_107		:DINT;
	Nr_108		:DINT;
	Nr_109		:DINT;
	Nr_110		:DINT;
	Nr_111		:DINT;
	Nr_112		:DINT;
	Nr_113		:DINT;
	Nr_114		:DINT;
	Nr_115		:DINT;
	Nr_116		:DINT;
	Nr_117		:DINT;
	Nr_118		:DINT;
	Nr_119		:DINT;
	Nr_120		:DINT;
	Nr_121		:DINT;
	Nr_122		:DINT;
	Nr_123		:DINT;
	Nr_124		:DINT;
	Nr_125		:DINT;
	Nr_126		:DINT;
	Nr_127		:DINT;
	Nr_128		:DINT;
	Nr_129		:DINT;
	Nr_130		:DINT;
	Nr_131		:DINT;
	Nr_132		:DINT;
	Nr_133		:DINT;
	Nr_134		:DINT;
	Nr_135		:DINT;
	Nr_136		:DINT;
	Nr_137		:DINT;
	Nr_138		:DINT;
	Nr_139		:DINT;
	Nr_140		:DINT;
	Nr_141		:DINT;
	Nr_142		:DINT;
	Nr_143		:DINT;
	Nr_144		:DINT;
	Nr_145		:DINT;
	Nr_146		:DINT;
	Nr_147		:DINT;
	Nr_148		:DINT;
	Nr_149		:DINT;
	Nr_150		:DINT;
	Nr_151		:DINT;
	Nr_152		:DINT;
	Nr_153		:DINT;
	Nr_154		:DINT;
	Nr_155		:DINT;
	Nr_156		:DINT;
	Nr_157		:DINT;
	Nr_158		:DINT;
	Nr_159		:DINT;
	Nr_160		:DINT;
	Nr_161		:DINT;
	Nr_162		:DINT;
	Nr_163		:DINT;
	Nr_164		:DINT;
	Nr_165		:DINT;
	Nr_166		:DINT;
	Nr_167		:DINT;
	Nr_168		:DINT;
	Nr_169		:DINT;
	Nr_170		:DINT;
	Nr_171		:DINT;
	Nr_172		:DINT;
	Nr_173		:DINT;
	Nr_174		:DINT;
	Nr_175		:DINT;
	Nr_176		:DINT;
	Nr_177		:DINT;
	Nr_178		:DINT;
	Nr_179		:DINT;
	Nr_180		:DINT;
	Nr_181		:DINT;
	Nr_182		:DINT;
	Nr_183		:DINT;
	Nr_184		:DINT;
	Nr_185		:DINT;
	Nr_186		:DINT;
	Nr_187		:DINT;
	Nr_188		:DINT;
	Nr_189		:DINT;
	Nr_190		:DINT;
	Nr_191		:DINT;
	Nr_192		:DINT;
	Nr_193		:DINT;
	Nr_194		:DINT;
	Nr_195		:DINT;
	Nr_196		:DINT;
	Nr_197		:DINT;
	Nr_198		:DINT;
	Nr_199		:DINT;
	
END_STRUCT
END_TYPE

// ---- SRT_Allgemein/0010_Bausteine_mitDuts/DUTs/Meldungen/DUT_Meldungen_0000.TcDUT
TYPE DUT_Meldungen_0000 :
STRUCT
					  // #MText: Achtung ein Fehler #HText: Achtung eine Hilfe #Prio: 1-10 Error 11-20 Warnung 21-30 Info #BMK:	

	Nr_001		:BOOL;// #MText: #HText: #Prio: #BMK:
	Nr_002		:BOOL;// #MText: #HText: #Prio: #BMK: 
	Nr_003		:BOOL;// #MText: #HText: #Prio: #BMK: 
	Nr_004		:BOOL;// #MText: #HText: #Prio: #BMK: 
	Nr_005		:BOOL;// #MText: #HText: #Prio: #BMK: 
	Nr_006		:BOOL;// #MText: #HText: #Prio: #BMK: 
	Nr_007		:BOOL;// #MText: #HText: #Prio: #BMK: 
	Nr_008		:BOOL;// #MText: #HText: #Prio: #BMK: 
	Nr_009		:BOOL;// #MText: #HText: #Prio: #BMK: 
	Nr_010		:BOOL;// #MText: #HText: #Prio: #BMK: 
	Nr_011		:BOOL;// #MText: #HText: #Prio: #BMK: 
	Nr_012		:BOOL;// #MText: #HText: #Prio: #BMK: 
	Nr_013		:BOOL;// #MText: #HText: #Prio: #BMK: 
	Nr_014		:BOOL;// #MText: #HText: #Prio: #BMK: 
	Nr_015		:BOOL;// #MText: #HText: #Prio: #BMK:     
	Nr_016		:BOOL;// #MText: #HText: #Prio: #BMK:
	Nr_017		:BOOL;// #MText: #HText: #Prio: #BMK:     
	Nr_018		:BOOL;// #MText: #HText: #Prio: #BMK:
	Nr_019		:BOOL;// #MText: #HText: #Prio: #BMK:     
	Nr_020		:BOOL;// #MText: #HText: #Prio: #BMK:
	Nr_021		:BOOL;// #MText: #HText: #Prio: #BMK:     
	Nr_022		:BOOL;// #MText: #HText: #Prio: #BMK:     
	Nr_023		:BOOL;// #MText: #HText: #Prio: #BMK:      
	Nr_024		:BOOL;// #MText: #HText: #Prio: #BMK:
	Nr_025		:BOOL;// #MText: #HText: #Prio: #BMK:      
	Nr_026		:BOOL;// #MText: #HText: #Prio: #BMK:
	Nr_027		:BOOL;// #MText: #HText: #Prio: #BMK:      
	Nr_028		:BOOL;// #MText: #HText: #Prio: #BMK:
	Nr_029		:BOOL;// #MText: #HText: #Prio: #BMK:      
	Nr_030		:BOOL;// #MText: #HText: #Prio: #BMK:
	Nr_031		:BOOL;// #MText: #HText: #Prio: #BMK:      
	Nr_032		:BOOL;// #MText: #HText: #Prio: #BMK:
	Nr_033		:BOOL;// #MText: #HText: #Prio: #BMK:      
	Nr_034		:BOOL;// #MText: #HText: #Prio: #BMK:
	Nr_035		:BOOL;// #MText: #HText: #Prio: #BMK:      
	Nr_036		:BOOL;// #MText: #HText: #Prio: #BMK:
	Nr_037		:BOOL;// #MText: #HText: #Prio: #BMK:
	Nr_038		:BOOL;// #MText: #HText: #Prio: #BMK:
	Nr_039		:BOOL;// #MText: #HText: #Prio: #BMK:
	Nr_040		:BOOL;// #MText: #HText: #Prio: #BMK:
	Nr_041		:BOOL;// #MText: #HText: #Prio: #BMK:
	Nr_042		:BOOL;// #MText: #HText: #Prio: #BMK:
	Nr_043		:BOOL;// #MText: #HText: #Prio: #BMK:
	Nr_044		:BOOL;// #MText: #HText: #Prio: #BMK:
	Nr_045		:BOOL;// #MText: #HText: #Prio: #BMK:
	Nr_046		:BOOL;// #MText: #HText: #Prio: #BMK:
	Nr_047		:BOOL;// #MText: #HText: #Prio: #BMK:
	Nr_048		:BOOL;// #MText: #HText: #Prio: #BMK:
	Nr_049		:BOOL;// #MText: #HText: #Prio: #BMK:
	Nr_050		:BOOL;// #MText: #HText: #Prio: #BMK:
	Nr_051		:BOOL;// #MText: #HText: #Prio: #BMK:
	Nr_052		:BOOL;// #MText: #HText: #Prio: #BMK:
	Nr_053		:BOOL;// #MText: #HText: #Prio: #BMK:
	Nr_054		:BOOL;// #MText: #HText: #Prio: #BMK:
	Nr_055		:BOOL;// #MText: #HText: #Prio: #BMK:
	Nr_056		:BOOL;// #MText: #HText: #Prio: #BMK:
	Nr_057		:BOOL;// #MText: #HText: #Prio: #BMK:
	Nr_058		:BOOL;// #MText: #HText: #Prio: #BMK:
	Nr_059		:BOOL;// #MText: #HText: #Prio: #BMK:
	Nr_060		:BOOL;// #MText: #HText: #Prio: #BMK:
	Nr_061		:BOOL;// #MText: #HText: #Prio: #BMK:
	Nr_062		:BOOL;// #MText: #HText: #Prio: #BMK:
	Nr_063		:BOOL;// #MText: #HText: #Prio: #BMK:
	Nr_064		:BOOL;// #MText: #HText: #Prio: #BMK:
	Nr_065		:BOOL;// #MText: #HText: #Prio: #BMK:
	Nr_066		:BOOL;// #MText: #HText: #Prio: #BMK:
	Nr_067		:BOOL;// #MText: #HText: #Prio: #BMK:
	Nr_068		:BOOL;// #MText: #HText: #Prio: #BMK:
	Nr_069		:BOOL;// #MText: #HText: #Prio: #BMK:
	Nr_070		:BOOL;// #MText: #HText: #Prio: #BMK:
	Nr_071		:BOOL;// #MText: #HText: #Prio: #BMK:
	Nr_072		:BOOL;// #MText: #HText: #Prio: #BMK:
	Nr_073		:BOOL;// #MText: #HText: #Prio: #BMK:
	Nr_074		:BOOL;// #MText: #HText: #Prio: #BMK:
	Nr_075		:BOOL;// #MText: #HText: #Prio: #BMK:
	Nr_076		:BOOL;// #MText: #HText: #Prio: #BMK:
	Nr_077		:BOOL;// #MText: #HText: #Prio: #BMK:
	Nr_078		:BOOL;// #MText: #HText: #Prio: #BMK:
	Nr_079		:BOOL;// #MText: #HText: #Prio: #BMK:
	Nr_080		:BOOL;// #MText: #HText: #Prio: #BMK:
	Nr_081		:BOOL;// #MText: #HText: #Prio: #BMK:
	Nr_082		:BOOL;// #MText: #HText: #Prio: #BMK:
	Nr_083		:BOOL;// #MText: #HText: #Prio: #BMK:
	Nr_084		:BOOL;// #MText: #HText: #Prio: #BMK:
	Nr_085		:BOOL;// #MText: #HText: #Prio: #BMK:
	Nr_086		:BOOL;// #MText: #HText: #Prio: #BMK:
	Nr_087		:BOOL;// #MText: #HText: #Prio: #BMK:
	Nr_088		:BOOL;// #MText: #HText: #Prio: #BMK:
	Nr_089		:BOOL;// #MText: #HText: #Prio: #BMK:
	Nr_090		:BOOL;// #MText: #HText: #Prio: #BMK:
	Nr_091		:BOOL;// #MText: #HText: #Prio: #BMK:
	Nr_092		:BOOL;// #MText: #HText: #Prio: #BMK:
	Nr_093		:BOOL;// #MText: #HText: #Prio: #BMK:
	Nr_094		:BOOL;// #MText: #HText: #Prio: #BMK:
	Nr_095		:BOOL;// #MText: #HText: #Prio: #BMK:
	Nr_096		:BOOL;// #MText: #HText: #Prio: #BMK:
	Nr_097		:BOOL;// #MText: #HText: #Prio: #BMK:
	Nr_098		:BOOL;// #MText: #HText: #Prio: #BMK:
	Nr_099		:BOOL;// #MText: #HText: #Prio: #BMK:
	
	Nr_100		:BOOL;// #MText: #HText: #Prio: #BMK:
	Nr_101		:BOOL;// #MText: #HText: #Prio: #BMK:
	Nr_102		:BOOL;// #MText: #HText: #Prio: #BMK:
	Nr_103		:BOOL;// #MText: #HText: #Prio: #BMK:
	Nr_104		:BOOL;// #MText: #HText: #Prio: #BMK:
	Nr_105		:BOOL;// #MText: #HText: #Prio: #BMK:
	Nr_106		:BOOL;// #MText: #HText: #Prio: #BMK:
	Nr_107		:BOOL;// #MText: #HText: #Prio: #BMK:
	Nr_108		:BOOL;// #MText: #HText: #Prio: #BMK:
	Nr_109		:BOOL;// #MText: #HText: #Prio: #BMK:
	Nr_110		:BOOL;// #MText: #HText: #Prio: #BMK:
	Nr_111		:BOOL;// #MText: #HText: #Prio: #BMK:
	Nr_112		:BOOL;// #MText: #HText: #Prio: #BMK:
	Nr_113		:BOOL;// #MText: #HText: #Prio: #BMK:
	Nr_114		:BOOL;// #MText: #HText: #Prio: #BMK:
	Nr_115		:BOOL;// #MText: #HText: #Prio: #BMK:
	Nr_116		:BOOL;// #MText: #HText: #Prio: #BMK:
	Nr_117		:BOOL;// #MText: #HText: #Prio: #BMK:
	Nr_118		:BOOL;// #MText: #HText: #Prio: #BMK:
	Nr_119		:BOOL;// #MText: #HText: #Prio: #BMK:
	Nr_120		:BOOL;// #MText: #HText: #Prio: #BMK:
	Nr_121		:BOOL;// #MText: #HText: #Prio: #BMK:
	Nr_122		:BOOL;// #MText: #HText: #Prio: #BMK:
	Nr_123		:BOOL;// #MText: #HText: #Prio: #BMK:
	Nr_124		:BOOL;// #MText: #HText: #Prio: #BMK:
	Nr_125		:BOOL;// #MText: #HText: #Prio: #BMK:
	Nr_126		:BOOL;// #MText: #HText: #Prio: #BMK:
	Nr_127		:BOOL;// #MText: #HText: #Prio: #BMK:
	Nr_128		:BOOL;// #MText: #HText: #Prio: #BMK:
	Nr_129		:BOOL;// #MText: #HText: #Prio: #BMK:
	Nr_130		:BOOL;// #MText: #HText: #Prio: #BMK:
	Nr_131		:BOOL;// #MText: #HText: #Prio: #BMK:
	Nr_132		:BOOL;// #MText: #HText: #Prio: #BMK:
	Nr_133		:BOOL;// #MText: #HText: #Prio: #BMK:
	Nr_134		:BOOL;// #MText: #HText: #Prio: #BMK:
	Nr_135		:BOOL;// #MText: #HText: #Prio: #BMK:
	Nr_136		:BOOL;// #MText: #HText: #Prio: #BMK:
	Nr_137		:BOOL;// #MText: #HText: #Prio: #BMK:
	Nr_138		:BOOL;// #MText: #HText: #Prio: #BMK:
	Nr_139		:BOOL;// #MText: #HText: #Prio: #BMK:
	Nr_140		:BOOL;// #MText: #HText: #Prio: #BMK:
	Nr_141		:BOOL;// #MText: #HText: #Prio: #BMK:
	Nr_142		:BOOL;// #MText: #HText: #Prio: #BMK:
	Nr_143		:BOOL;// #MText: #HText: #Prio: #BMK:
	Nr_144		:BOOL;// #MText: #HText: #Prio: #BMK:
	Nr_145		:BOOL;// #MText: #HText: #Prio: #BMK:
	Nr_146		:BOOL;// #MText: #HText: #Prio: #BMK:
	Nr_147		:BOOL;// #MText: #HText: #Prio: #BMK:
	Nr_148		:BOOL;// #MText: #HText: #Prio: #BMK:
	Nr_149		:BOOL;// #MText: #HText: #Prio: #BMK:
	Nr_150		:BOOL;// #MText: #HText: #Prio: #BMK:
	Nr_151		:BOOL;// #MText: #HText: #Prio: #BMK:
	Nr_152		:BOOL;// #MText: #HText: #Prio: #BMK:
	Nr_153		:BOOL;// #MText: #HText: #Prio: #BMK:
	Nr_154		:BOOL;// #MText: #HText: #Prio: #BMK:
	Nr_155		:BOOL;// #MText: #HText: #Prio: #BMK:
	Nr_156		:BOOL;// #MText: #HText: #Prio: #BMK:
	Nr_157		:BOOL;// #MText: #HText: #Prio: #BMK:
	Nr_158		:BOOL;// #MText: #HText: #Prio: #BMK:
	Nr_159		:BOOL;// #MText: #HText: #Prio: #BMK:
	Nr_160		:BOOL;// #MText: #HText: #Prio: #BMK:
	Nr_161		:BOOL;// #MText: #HText: #Prio: #BMK:
	Nr_162		:BOOL;// #MText: #HText: #Prio: #BMK:
	Nr_163		:BOOL;// #MText: #HText: #Prio: #BMK:
	Nr_164		:BOOL;// #MText: #HText: #Prio: #BMK:
	Nr_165		:BOOL;// #MText: #HText: #Prio: #BMK:
	Nr_166		:BOOL;// #MText: #HText: #Prio: #BMK:
	Nr_167		:BOOL;// #MText: #HText: #Prio: #BMK:
	Nr_168		:BOOL;// #MText: #HText: #Prio: #BMK:
	Nr_169		:BOOL;// #MText: #HText: #Prio: #BMK:
	Nr_170		:BOOL;// #MText: #HText: #Prio: #BMK:
	Nr_171		:BOOL;// #MText: #HText: #Prio: #BMK:
	Nr_172		:BOOL;// #MText: #HText: #Prio: #BMK:
	Nr_173		:BOOL;// #MText: #HText: #Prio: #BMK:
	Nr_174		:BOOL;// #MText: #HText: #Prio: #BMK:
	Nr_175		:BOOL;// #MText: #HText: #Prio: #BMK:
	Nr_176		:BOOL;// #MText: #HText: #Prio: #BMK:
	Nr_177		:BOOL;// #MText: #HText: #Prio: #BMK:
	Nr_178		:BOOL;// #MText: #HText: #Prio: #BMK:
	Nr_179		:BOOL;// #MText: #HText: #Prio: #BMK:
	Nr_180		:BOOL;// #MText: #HText: #Prio: #BMK:
	Nr_181		:BOOL;// #MText: #HText: #Prio: #BMK:
	Nr_182		:BOOL;// #MText: #HText: #Prio: #BMK:
	Nr_183		:BOOL;// #MText: #HText: #Prio: #BMK:
	Nr_184		:BOOL;// #MText: #HText: #Prio: #BMK:
	Nr_185		:BOOL;// #MText: #HText: #Prio: #BMK:
	Nr_186		:BOOL;// #MText: #HText: #Prio: #BMK:
	Nr_187		:BOOL;// #MText: #HText: #Prio: #BMK:
	Nr_188		:BOOL;// #MText: #HText: #Prio: #BMK:
	Nr_189		:BOOL;// #MText: #HText: #Prio: #BMK:
	Nr_190		:BOOL;// #MText: #HText: #Prio: #BMK:
	Nr_191		:BOOL;// #MText: #HText: #Prio: #BMK:
	Nr_192		:BOOL;// #MText: #HText: #Prio: #BMK:
	Nr_193		:BOOL;// #MText: #HText: #Prio: #BMK:
	Nr_194		:BOOL;// #MText: #HText: #Prio: #BMK:
	Nr_195		:BOOL;// #MText: #HText: #Prio: #BMK:
	Nr_196		:BOOL;// #MText: #HText: #Prio: #BMK:
	Nr_197		:BOOL;// #MText: #HText: #Prio: #BMK:
	Nr_198		:BOOL;// #MText: #HText: #Prio: #BMK:
	Nr_199		:BOOL;// #MText: #HText: #Prio: #BMK:
	
END_STRUCT
END_TYPE

// ---- SRT_Allgemein/0010_Bausteine_mitDuts/DUTs/Meldungen/DUT_Meldungen_1000.TcDUT
TYPE DUT_Meldungen_1000 :
STRUCT
					  // #MText: Achtung ein Fehler #HText: Achtung eine Hilfe #Prio: 1-10 Error 11-20 Warnung 21-30 Info #BMK:	

	Nr_001		:BOOL;// #MText: #HText: #Prio: #BMK:
	Nr_002		:BOOL;// #MText: #HText: #Prio: #BMK: 
	Nr_003		:BOOL;// #MText: #HText: #Prio: #BMK: 
	Nr_004		:BOOL;// #MText: #HText: #Prio: #BMK: 
	Nr_005		:BOOL;// #MText: #HText: #Prio: #BMK: 
	Nr_006		:BOOL;// #MText: #HText: #Prio: #BMK: 
	Nr_007		:BOOL;// #MText: #HText: #Prio: #BMK: 
	Nr_008		:BOOL;// #MText: #HText: #Prio: #BMK: 
	Nr_009		:BOOL;// #MText: #HText: #Prio: #BMK: 
	Nr_010		:BOOL;// #MText: #HText: #Prio: #BMK: 
	Nr_011		:BOOL;// #MText: #HText: #Prio: #BMK: 
	Nr_012		:BOOL;// #MText: #HText: #Prio: #BMK: 
	Nr_013		:BOOL;// #MText: #HText: #Prio: #BMK: 
	Nr_014		:BOOL;// #MText: #HText: #Prio: #BMK: 
	Nr_015		:BOOL;// #MText: #HText: #Prio: #BMK:     
	Nr_016		:BOOL;// #MText: #HText: #Prio: #BMK:
	Nr_017		:BOOL;// #MText: #HText: #Prio: #BMK:     
	Nr_018		:BOOL;// #MText: #HText: #Prio: #BMK:
	Nr_019		:BOOL;// #MText: #HText: #Prio: #BMK:     
	Nr_020		:BOOL;// #MText: #HText: #Prio: #BMK:
	Nr_021		:BOOL;// #MText: #HText: #Prio: #BMK:     
	Nr_022		:BOOL;// #MText: #HText: #Prio: #BMK:     
	Nr_023		:BOOL;// #MText: #HText: #Prio: #BMK:      
	Nr_024		:BOOL;// #MText: #HText: #Prio: #BMK:
	Nr_025		:BOOL;// #MText: #HText: #Prio: #BMK:      
	Nr_026		:BOOL;// #MText: #HText: #Prio: #BMK:
	Nr_027		:BOOL;// #MText: #HText: #Prio: #BMK:      
	Nr_028		:BOOL;// #MText: #HText: #Prio: #BMK:
	Nr_029		:BOOL;// #MText: #HText: #Prio: #BMK:      
	Nr_030		:BOOL;// #MText: #HText: #Prio: #BMK:
	Nr_031		:BOOL;// #MText: #HText: #Prio: #BMK:      
	Nr_032		:BOOL;// #MText: #HText: #Prio: #BMK:
	Nr_033		:BOOL;// #MText: #HText: #Prio: #BMK:      
	Nr_034		:BOOL;// #MText: #HText: #Prio: #BMK:
	Nr_035		:BOOL;// #MText: #HText: #Prio: #BMK:      
	Nr_036		:BOOL;// #MText: #HText: #Prio: #BMK:
	Nr_037		:BOOL;// #MText: #HText: #Prio: #BMK:
	Nr_038		:BOOL;// #MText: #HText: #Prio: #BMK:
	Nr_039		:BOOL;// #MText: #HText: #Prio: #BMK:
	Nr_040		:BOOL;// #MText: #HText: #Prio: #BMK:
	Nr_041		:BOOL;// #MText: #HText: #Prio: #BMK:
	Nr_042		:BOOL;// #MText: #HText: #Prio: #BMK:
	Nr_043		:BOOL;// #MText: #HText: #Prio: #BMK:
	Nr_044		:BOOL;// #MText: #HText: #Prio: #BMK:
	Nr_045		:BOOL;// #MText: #HText: #Prio: #BMK:
	Nr_046		:BOOL;// #MText: #HText: #Prio: #BMK:
	Nr_047		:BOOL;// #MText: #HText: #Prio: #BMK:
	Nr_048		:BOOL;// #MText: #HText: #Prio: #BMK:
	Nr_049		:BOOL;// #MText: #HText: #Prio: #BMK:
	Nr_050		:BOOL;// #MText: #HText: #Prio: #BMK:
	Nr_051		:BOOL;// #MText: #HText: #Prio: #BMK:
	Nr_052		:BOOL;// #MText: #HText: #Prio: #BMK:
	Nr_053		:BOOL;// #MText: #HText: #Prio: #BMK:
	Nr_054		:BOOL;// #MText: #HText: #Prio: #BMK:
	Nr_055		:BOOL;// #MText: #HText: #Prio: #BMK:
	Nr_056		:BOOL;// #MText: #HText: #Prio: #BMK:
	Nr_057		:BOOL;// #MText: #HText: #Prio: #BMK:
	Nr_058		:BOOL;// #MText: #HText: #Prio: #BMK:
	Nr_059		:BOOL;// #MText: #HText: #Prio: #BMK:
	Nr_060		:BOOL;// #MText: #HText: #Prio: #BMK:
	Nr_061		:BOOL;// #MText: #HText: #Prio: #BMK:
	Nr_062		:BOOL;// #MText: #HText: #Prio: #BMK:
	Nr_063		:BOOL;// #MText: #HText: #Prio: #BMK:
	Nr_064		:BOOL;// #MText: #HText: #Prio: #BMK:
	Nr_065		:BOOL;// #MText: #HText: #Prio: #BMK:
	Nr_066		:BOOL;// #MText: #HText: #Prio: #BMK:
	Nr_067		:BOOL;// #MText: #HText: #Prio: #BMK:
	Nr_068		:BOOL;// #MText: #HText: #Prio: #BMK:
	Nr_069		:BOOL;// #MText: #HText: #Prio: #BMK:
	Nr_070		:BOOL;// #MText: #HText: #Prio: #BMK:
	Nr_071		:BOOL;// #MText: #HText: #Prio: #BMK:
	Nr_072		:BOOL;// #MText: #HText: #Prio: #BMK:
	Nr_073		:BOOL;// #MText: #HText: #Prio: #BMK:
	Nr_074		:BOOL;// #MText: #HText: #Prio: #BMK:
	Nr_075		:BOOL;// #MText: #HText: #Prio: #BMK:
	Nr_076		:BOOL;// #MText: #HText: #Prio: #BMK:
	Nr_077		:BOOL;// #MText: #HText: #Prio: #BMK:
	Nr_078		:BOOL;// #MText: #HText: #Prio: #BMK:
	Nr_079		:BOOL;// #MText: #HText: #Prio: #BMK:
	Nr_080		:BOOL;// #MText: #HText: #Prio: #BMK:
	Nr_081		:BOOL;// #MText: #HText: #Prio: #BMK:
	Nr_082		:BOOL;// #MText: #HText: #Prio: #BMK:
	Nr_083		:BOOL;// #MText: #HText: #Prio: #BMK:
	Nr_084		:BOOL;// #MText: #HText: #Prio: #BMK:
	Nr_085		:BOOL;// #MText: #HText: #Prio: #BMK:
	Nr_086		:BOOL;// #MText: #HText: #Prio: #BMK:
	Nr_087		:BOOL;// #MText: #HText: #Prio: #BMK:
	Nr_088		:BOOL;// #MText: #HText: #Prio: #BMK:
	Nr_089		:BOOL;// #MText: #HText: #Prio: #BMK:
	Nr_090		:BOOL;// #MText: #HText: #Prio: #BMK:
	Nr_091		:BOOL;// #MText: #HText: #Prio: #BMK:
	Nr_092		:BOOL;// #MText: #HText: #Prio: #BMK:
	Nr_093		:BOOL;// #MText: #HText: #Prio: #BMK:
	Nr_094		:BOOL;// #MText: #HText: #Prio: #BMK:
	Nr_095		:BOOL;// #MText: #HText: #Prio: #BMK:
	Nr_096		:BOOL;// #MText: #HText: #Prio: #BMK:
	Nr_097		:BOOL;// #MText: #HText: #Prio: #BMK:
	Nr_098		:BOOL;// #MText: #HText: #Prio: #BMK:
	Nr_099		:BOOL;// #MText: #HText: #Prio: #BMK:
	
	Nr_100		:BOOL;// #MText: #HText: #Prio: #BMK:
	Nr_101		:BOOL;// #MText: #HText: #Prio: #BMK:
	Nr_102		:BOOL;// #MText: #HText: #Prio: #BMK:
	Nr_103		:BOOL;// #MText: #HText: #Prio: #BMK:
	Nr_104		:BOOL;// #MText: #HText: #Prio: #BMK:
	Nr_105		:BOOL;// #MText: #HText: #Prio: #BMK:
	Nr_106		:BOOL;// #MText: #HText: #Prio: #BMK:
	Nr_107		:BOOL;// #MText: #HText: #Prio: #BMK:
	Nr_108		:BOOL;// #MText: #HText: #Prio: #BMK:
	Nr_109		:BOOL;// #MText: #HText: #Prio: #BMK:
	Nr_110		:BOOL;// #MText: #HText: #Prio: #BMK:
	Nr_111		:BOOL;// #MText: #HText: #Prio: #BMK:
	Nr_112		:BOOL;// #MText: #HText: #Prio: #BMK:
	Nr_113		:BOOL;// #MText: #HText: #Prio: #BMK:
	Nr_114		:BOOL;// #MText: #HText: #Prio: #BMK:
	Nr_115		:BOOL;// #MText: #HText: #Prio: #BMK:
	Nr_116		:BOOL;// #MText: #HText: #Prio: #BMK:
	Nr_117		:BOOL;// #MText: #HText: #Prio: #BMK:
	Nr_118		:BOOL;// #MText: #HText: #Prio: #BMK:
	Nr_119		:BOOL;// #MText: #HText: #Prio: #BMK:
	Nr_120		:BOOL;// #MText: #HText: #Prio: #BMK:
	Nr_121		:BOOL;// #MText: #HText: #Prio: #BMK:
	Nr_122		:BOOL;// #MText: #HText: #Prio: #BMK:
	Nr_123		:BOOL;// #MText: #HText: #Prio: #BMK:
	Nr_124		:BOOL;// #MText: #HText: #Prio: #BMK:
	Nr_125		:BOOL;// #MText: #HText: #Prio: #BMK:
	Nr_126		:BOOL;// #MText: #HText: #Prio: #BMK:
	Nr_127		:BOOL;// #MText: #HText: #Prio: #BMK:
	Nr_128		:BOOL;// #MText: #HText: #Prio: #BMK:
	Nr_129		:BOOL;// #MText: #HText: #Prio: #BMK:
	Nr_130		:BOOL;// #MText: #HText: #Prio: #BMK:
	Nr_131		:BOOL;// #MText: #HText: #Prio: #BMK:
	Nr_132		:BOOL;// #MText: #HText: #Prio: #BMK:
	Nr_133		:BOOL;// #MText: #HText: #Prio: #BMK:
	Nr_134		:BOOL;// #MText: #HText: #Prio: #BMK:
	Nr_135		:BOOL;// #MText: #HText: #Prio: #BMK:
	Nr_136		:BOOL;// #MText: #HText: #Prio: #BMK:
	Nr_137		:BOOL;// #MText: #HText: #Prio: #BMK:
	Nr_138		:BOOL;// #MText: #HText: #Prio: #BMK:
	Nr_139		:BOOL;// #MText: #HText: #Prio: #BMK:
	Nr_140		:BOOL;// #MText: #HText: #Prio: #BMK:
	Nr_141		:BOOL;// #MText: #HText: #Prio: #BMK:
	Nr_142		:BOOL;// #MText: #HText: #Prio: #BMK:
	Nr_143		:BOOL;// #MText: #HText: #Prio: #BMK:
	Nr_144		:BOOL;// #MText: #HText: #Prio: #BMK:
	Nr_145		:BOOL;// #MText: #HText: #Prio: #BMK:
	Nr_146		:BOOL;// #MText: #HText: #Prio: #BMK:
	Nr_147		:BOOL;// #MText: #HText: #Prio: #BMK:
	Nr_148		:BOOL;// #MText: #HText: #Prio: #BMK:
	Nr_149		:BOOL;// #MText: #HText: #Prio: #BMK:
	Nr_150		:BOOL;// #MText: #HText: #Prio: #BMK:
	Nr_151		:BOOL;// #MText: #HText: #Prio: #BMK:
	Nr_152		:BOOL;// #MText: #HText: #Prio: #BMK:
	Nr_153		:BOOL;// #MText: #HText: #Prio: #BMK:
	Nr_154		:BOOL;// #MText: #HText: #Prio: #BMK:
	Nr_155		:BOOL;// #MText: #HText: #Prio: #BMK:
	Nr_156		:BOOL;// #MText: #HText: #Prio: #BMK:
	Nr_157		:BOOL;// #MText: #HText: #Prio: #BMK:
	Nr_158		:BOOL;// #MText: #HText: #Prio: #BMK:
	Nr_159		:BOOL;// #MText: #HText: #Prio: #BMK:
	Nr_160		:BOOL;// #MText: #HText: #Prio: #BMK:
	Nr_161		:BOOL;// #MText: #HText: #Prio: #BMK:
	Nr_162		:BOOL;// #MText: #HText: #Prio: #BMK:
	Nr_163		:BOOL;// #MText: #HText: #Prio: #BMK:
	Nr_164		:BOOL;// #MText: #HText: #Prio: #BMK:
	Nr_165		:BOOL;// #MText: #HText: #Prio: #BMK:
	Nr_166		:BOOL;// #MText: #HText: #Prio: #BMK:
	Nr_167		:BOOL;// #MText: #HText: #Prio: #BMK:
	Nr_168		:BOOL;// #MText: #HText: #Prio: #BMK:
	Nr_169		:BOOL;// #MText: #HText: #Prio: #BMK:
	Nr_170		:BOOL;// #MText: #HText: #Prio: #BMK:
	Nr_171		:BOOL;// #MText: #HText: #Prio: #BMK:
	Nr_172		:BOOL;// #MText: #HText: #Prio: #BMK:
	Nr_173		:BOOL;// #MText: #HText: #Prio: #BMK:
	Nr_174		:BOOL;// #MText: #HText: #Prio: #BMK:
	Nr_175		:BOOL;// #MText: #HText: #Prio: #BMK:
	Nr_176		:BOOL;// #MText: #HText: #Prio: #BMK:
	Nr_177		:BOOL;// #MText: #HText: #Prio: #BMK:
	Nr_178		:BOOL;// #MText: #HText: #Prio: #BMK:
	Nr_179		:BOOL;// #MText: #HText: #Prio: #BMK:
	Nr_180		:BOOL;// #MText: #HText: #Prio: #BMK:
	Nr_181		:BOOL;// #MText: #HText: #Prio: #BMK:
	Nr_182		:BOOL;// #MText: #HText: #Prio: #BMK:
	Nr_183		:BOOL;// #MText: #HText: #Prio: #BMK:
	Nr_184		:BOOL;// #MText: #HText: #Prio: #BMK:
	Nr_185		:BOOL;// #MText: #HText: #Prio: #BMK:
	Nr_186		:BOOL;// #MText: #HText: #Prio: #BMK:
	Nr_187		:BOOL;// #MText: #HText: #Prio: #BMK:
	Nr_188		:BOOL;// #MText: #HText: #Prio: #BMK:
	Nr_189		:BOOL;// #MText: #HText: #Prio: #BMK:
	Nr_190		:BOOL;// #MText: #HText: #Prio: #BMK:
	Nr_191		:BOOL;// #MText: #HText: #Prio: #BMK:
	Nr_192		:BOOL;// #MText: #HText: #Prio: #BMK:
	Nr_193		:BOOL;// #MText: #HText: #Prio: #BMK:
	Nr_194		:BOOL;// #MText: #HText: #Prio: #BMK:
	Nr_195		:BOOL;// #MText: #HText: #Prio: #BMK:
	Nr_196		:BOOL;// #MText: #HText: #Prio: #BMK:
	Nr_197		:BOOL;// #MText: #HText: #Prio: #BMK:
	Nr_198		:BOOL;// #MText: #HText: #Prio: #BMK:
	Nr_199		:BOOL;// #MText: #HText: #Prio: #BMK:
	
END_STRUCT
END_TYPE

// ---- SRT_Allgemein/0010_Bausteine_mitDuts/DUTs/Meldungen/DUT_Meldungen_2000.TcDUT
TYPE DUT_Meldungen_2000 :
STRUCT
					  // #MText: Achtung ein Fehler #HText: Achtung eine Hilfe #Prio: 1-10 Error 11-20 Warnung 21-30 Info #BMK:	

	Nr_001		:BOOL;// #MText: #HText: #Prio: #BMK:
	Nr_002		:BOOL;// #MText: #HText: #Prio: #BMK: 
	Nr_003		:BOOL;// #MText: #HText: #Prio: #BMK: 
	Nr_004		:BOOL;// #MText: #HText: #Prio: #BMK: 
	Nr_005		:BOOL;// #MText: #HText: #Prio: #BMK: 
	Nr_006		:BOOL;// #MText: #HText: #Prio: #BMK: 
	Nr_007		:BOOL;// #MText: #HText: #Prio: #BMK: 
	Nr_008		:BOOL;// #MText: #HText: #Prio: #BMK: 
	Nr_009		:BOOL;// #MText: #HText: #Prio: #BMK: 
	Nr_010		:BOOL;// #MText: #HText: #Prio: #BMK: 
	Nr_011		:BOOL;// #MText: #HText: #Prio: #BMK: 
	Nr_012		:BOOL;// #MText: #HText: #Prio: #BMK: 
	Nr_013		:BOOL;// #MText: #HText: #Prio: #BMK: 
	Nr_014		:BOOL;// #MText: #HText: #Prio: #BMK: 
	Nr_015		:BOOL;// #MText: #HText: #Prio: #BMK:     
	Nr_016		:BOOL;// #MText: #HText: #Prio: #BMK:
	Nr_017		:BOOL;// #MText: #HText: #Prio: #BMK:     
	Nr_018		:BOOL;// #MText: #HText: #Prio: #BMK:
	Nr_019		:BOOL;// #MText: #HText: #Prio: #BMK:     
	Nr_020		:BOOL;// #MText: #HText: #Prio: #BMK:
	Nr_021		:BOOL;// #MText: #HText: #Prio: #BMK:     
	Nr_022		:BOOL;// #MText: #HText: #Prio: #BMK:     
	Nr_023		:BOOL;// #MText: #HText: #Prio: #BMK:      
	Nr_024		:BOOL;// #MText: #HText: #Prio: #BMK:
	Nr_025		:BOOL;// #MText: #HText: #Prio: #BMK:      
	Nr_026		:BOOL;// #MText: #HText: #Prio: #BMK:
	Nr_027		:BOOL;// #MText: #HText: #Prio: #BMK:      
	Nr_028		:BOOL;// #MText: #HText: #Prio: #BMK:
	Nr_029		:BOOL;// #MText: #HText: #Prio: #BMK:      
	Nr_030		:BOOL;// #MText: #HText: #Prio: #BMK:
	Nr_031		:BOOL;// #MText: #HText: #Prio: #BMK:      
	Nr_032		:BOOL;// #MText: #HText: #Prio: #BMK:
	Nr_033		:BOOL;// #MText: #HText: #Prio: #BMK:      
	Nr_034		:BOOL;// #MText: #HText: #Prio: #BMK:
	Nr_035		:BOOL;// #MText: #HText: #Prio: #BMK:      
	Nr_036		:BOOL;// #MText: #HText: #Prio: #BMK:
	Nr_037		:BOOL;// #MText: #HText: #Prio: #BMK:
	Nr_038		:BOOL;// #MText: #HText: #Prio: #BMK:
	Nr_039		:BOOL;// #MText: #HText: #Prio: #BMK:
	Nr_040		:BOOL;// #MText: #HText: #Prio: #BMK:
	Nr_041		:BOOL;// #MText: #HText: #Prio: #BMK:
	Nr_042		:BOOL;// #MText: #HText: #Prio: #BMK:
	Nr_043		:BOOL;// #MText: #HText: #Prio: #BMK:
	Nr_044		:BOOL;// #MText: #HText: #Prio: #BMK:
	Nr_045		:BOOL;// #MText: #HText: #Prio: #BMK:
	Nr_046		:BOOL;// #MText: #HText: #Prio: #BMK:
	Nr_047		:BOOL;// #MText: #HText: #Prio: #BMK:
	Nr_048		:BOOL;// #MText: #HText: #Prio: #BMK:
	Nr_049		:BOOL;// #MText: #HText: #Prio: #BMK:
	Nr_050		:BOOL;// #MText: #HText: #Prio: #BMK:
	Nr_051		:BOOL;// #MText: #HText: #Prio: #BMK:
	Nr_052		:BOOL;// #MText: #HText: #Prio: #BMK:
	Nr_053		:BOOL;// #MText: #HText: #Prio: #BMK:
	Nr_054		:BOOL;// #MText: #HText: #Prio: #BMK:
	Nr_055		:BOOL;// #MText: #HText: #Prio: #BMK:
	Nr_056		:BOOL;// #MText: #HText: #Prio: #BMK:
	Nr_057		:BOOL;// #MText: #HText: #Prio: #BMK:
	Nr_058		:BOOL;// #MText: #HText: #Prio: #BMK:
	Nr_059		:BOOL;// #MText: #HText: #Prio: #BMK:
	Nr_060		:BOOL;// #MText: #HText: #Prio: #BMK:
	Nr_061		:BOOL;// #MText: #HText: #Prio: #BMK:
	Nr_062		:BOOL;// #MText: #HText: #Prio: #BMK:
	Nr_063		:BOOL;// #MText: #HText: #Prio: #BMK:
	Nr_064		:BOOL;// #MText: #HText: #Prio: #BMK:
	Nr_065		:BOOL;// #MText: #HText: #Prio: #BMK:
	Nr_066		:BOOL;// #MText: #HText: #Prio: #BMK:
	Nr_067		:BOOL;// #MText: #HText: #Prio: #BMK:
	Nr_068		:BOOL;// #MText: #HText: #Prio: #BMK:
	Nr_069		:BOOL;// #MText: #HText: #Prio: #BMK:
	Nr_070		:BOOL;// #MText: #HText: #Prio: #BMK:
	Nr_071		:BOOL;// #MText: #HText: #Prio: #BMK:
	Nr_072		:BOOL;// #MText: #HText: #Prio: #BMK:
	Nr_073		:BOOL;// #MText: #HText: #Prio: #BMK:
	Nr_074		:BOOL;// #MText: #HText: #Prio: #BMK:
	Nr_075		:BOOL;// #MText: #HText: #Prio: #BMK:
	Nr_076		:BOOL;// #MText: #HText: #Prio: #BMK:
	Nr_077		:BOOL;// #MText: #HText: #Prio: #BMK:
	Nr_078		:BOOL;// #MText: #HText: #Prio: #BMK:
	Nr_079		:BOOL;// #MText: #HText: #Prio: #BMK:
	Nr_080		:BOOL;// #MText: #HText: #Prio: #BMK:
	Nr_081		:BOOL;// #MText: #HText: #Prio: #BMK:
	Nr_082		:BOOL;// #MText: #HText: #Prio: #BMK:
	Nr_083		:BOOL;// #MText: #HText: #Prio: #BMK:
	Nr_084		:BOOL;// #MText: #HText: #Prio: #BMK:
	Nr_085		:BOOL;// #MText: #HText: #Prio: #BMK:
	Nr_086		:BOOL;// #MText: #HText: #Prio: #BMK:
	Nr_087		:BOOL;// #MText: #HText: #Prio: #BMK:
	Nr_088		:BOOL;// #MText: #HText: #Prio: #BMK:
	Nr_089		:BOOL;// #MText: #HText: #Prio: #BMK:
	Nr_090		:BOOL;// #MText: #HText: #Prio: #BMK:
	Nr_091		:BOOL;// #MText: #HText: #Prio: #BMK:
	Nr_092		:BOOL;// #MText: #HText: #Prio: #BMK:
	Nr_093		:BOOL;// #MText: #HText: #Prio: #BMK:
	Nr_094		:BOOL;// #MText: #HText: #Prio: #BMK:
	Nr_095		:BOOL;// #MText: #HText: #Prio: #BMK:
	Nr_096		:BOOL;// #MText: #HText: #Prio: #BMK:
	Nr_097		:BOOL;// #MText: #HText: #Prio: #BMK:
	Nr_098		:BOOL;// #MText: #HText: #Prio: #BMK:
	Nr_099		:BOOL;// #MText: #HText: #Prio: #BMK:
	
	Nr_100		:BOOL;// #MText: #HText: #Prio: #BMK:
	Nr_101		:BOOL;// #MText: #HText: #Prio: #BMK:
	Nr_102		:BOOL;// #MText: #HText: #Prio: #BMK:
	Nr_103		:BOOL;// #MText: #HText: #Prio: #BMK:
	Nr_104		:BOOL;// #MText: #HText: #Prio: #BMK:
	Nr_105		:BOOL;// #MText: #HText: #Prio: #BMK:
	Nr_106		:BOOL;// #MText: #HText: #Prio: #BMK:
	Nr_107		:BOOL;// #MText: #HText: #Prio: #BMK:
	Nr_108		:BOOL;// #MText: #HText: #Prio: #BMK:
	Nr_109		:BOOL;// #MText: #HText: #Prio: #BMK:
	Nr_110		:BOOL;// #MText: #HText: #Prio: #BMK:
	Nr_111		:BOOL;// #MText: #HText: #Prio: #BMK:
	Nr_112		:BOOL;// #MText: #HText: #Prio: #BMK:
	Nr_113		:BOOL;// #MText: #HText: #Prio: #BMK:
	Nr_114		:BOOL;// #MText: #HText: #Prio: #BMK:
	Nr_115		:BOOL;// #MText: #HText: #Prio: #BMK:
	Nr_116		:BOOL;// #MText: #HText: #Prio: #BMK:
	Nr_117		:BOOL;// #MText: #HText: #Prio: #BMK:
	Nr_118		:BOOL;// #MText: #HText: #Prio: #BMK:
	Nr_119		:BOOL;// #MText: #HText: #Prio: #BMK:
	Nr_120		:BOOL;// #MText: #HText: #Prio: #BMK:
	Nr_121		:BOOL;// #MText: #HText: #Prio: #BMK:
	Nr_122		:BOOL;// #MText: #HText: #Prio: #BMK:
	Nr_123		:BOOL;// #MText: #HText: #Prio: #BMK:
	Nr_124		:BOOL;// #MText: #HText: #Prio: #BMK:
	Nr_125		:BOOL;// #MText: #HText: #Prio: #BMK:
	Nr_126		:BOOL;// #MText: #HText: #Prio: #BMK:
	Nr_127		:BOOL;// #MText: #HText: #Prio: #BMK:
	Nr_128		:BOOL;// #MText: #HText: #Prio: #BMK:
	Nr_129		:BOOL;// #MText: #HText: #Prio: #BMK:
	Nr_130		:BOOL;// #MText: #HText: #Prio: #BMK:
	Nr_131		:BOOL;// #MText: #HText: #Prio: #BMK:
	Nr_132		:BOOL;// #MText: #HText: #Prio: #BMK:
	Nr_133		:BOOL;// #MText: #HText: #Prio: #BMK:
	Nr_134		:BOOL;// #MText: #HText: #Prio: #BMK:
	Nr_135		:BOOL;// #MText: #HText: #Prio: #BMK:
	Nr_136		:BOOL;// #MText: #HText: #Prio: #BMK:
	Nr_137		:BOOL;// #MText: #HText: #Prio: #BMK:
	Nr_138		:BOOL;// #MText: #HText: #Prio: #BMK:
	Nr_139		:BOOL;// #MText: #HText: #Prio: #BMK:
	Nr_140		:BOOL;// #MText: #HText: #Prio: #BMK:
	Nr_141		:BOOL;// #MText: #HText: #Prio: #BMK:
	Nr_142		:BOOL;// #MText: #HText: #Prio: #BMK:
	Nr_143		:BOOL;// #MText: #HText: #Prio: #BMK:
	Nr_144		:BOOL;// #MText: #HText: #Prio: #BMK:
	Nr_145		:BOOL;// #MText: #HText: #Prio: #BMK:
	Nr_146		:BOOL;// #MText: #HText: #Prio: #BMK:
	Nr_147		:BOOL;// #MText: #HText: #Prio: #BMK:
	Nr_148		:BOOL;// #MText: #HText: #Prio: #BMK:
	Nr_149		:BOOL;// #MText: #HText: #Prio: #BMK:
	Nr_150		:BOOL;// #MText: #HText: #Prio: #BMK:
	Nr_151		:BOOL;// #MText: #HText: #Prio: #BMK:
	Nr_152		:BOOL;// #MText: #HText: #Prio: #BMK:
	Nr_153		:BOOL;// #MText: #HText: #Prio: #BMK:
	Nr_154		:BOOL;// #MText: #HText: #Prio: #BMK:
	Nr_155		:BOOL;// #MText: #HText: #Prio: #BMK:
	Nr_156		:BOOL;// #MText: #HText: #Prio: #BMK:
	Nr_157		:BOOL;// #MText: #HText: #Prio: #BMK:
	Nr_158		:BOOL;// #MText: #HText: #Prio: #BMK:
	Nr_159		:BOOL;// #MText: #HText: #Prio: #BMK:
	Nr_160		:BOOL;// #MText: #HText: #Prio: #BMK:
	Nr_161		:BOOL;// #MText: #HText: #Prio: #BMK:
	Nr_162		:BOOL;// #MText: #HText: #Prio: #BMK:
	Nr_163		:BOOL;// #MText: #HText: #Prio: #BMK:
	Nr_164		:BOOL;// #MText: #HText: #Prio: #BMK:
	Nr_165		:BOOL;// #MText: #HText: #Prio: #BMK:
	Nr_166		:BOOL;// #MText: #HText: #Prio: #BMK:
	Nr_167		:BOOL;// #MText: #HText: #Prio: #BMK:
	Nr_168		:BOOL;// #MText: #HText: #Prio: #BMK:
	Nr_169		:BOOL;// #MText: #HText: #Prio: #BMK:
	Nr_170		:BOOL;// #MText: #HText: #Prio: #BMK:
	Nr_171		:BOOL;// #MText: #HText: #Prio: #BMK:
	Nr_172		:BOOL;// #MText: #HText: #Prio: #BMK:
	Nr_173		:BOOL;// #MText: #HText: #Prio: #BMK:
	Nr_174		:BOOL;// #MText: #HText: #Prio: #BMK:
	Nr_175		:BOOL;// #MText: #HText: #Prio: #BMK:
	Nr_176		:BOOL;// #MText: #HText: #Prio: #BMK:
	Nr_177		:BOOL;// #MText: #HText: #Prio: #BMK:
	Nr_178		:BOOL;// #MText: #HText: #Prio: #BMK:
	Nr_179		:BOOL;// #MText: #HText: #Prio: #BMK:
	Nr_180		:BOOL;// #MText: #HText: #Prio: #BMK:
	Nr_181		:BOOL;// #MText: #HText: #Prio: #BMK:
	Nr_182		:BOOL;// #MText: #HText: #Prio: #BMK:
	Nr_183		:BOOL;// #MText: #HText: #Prio: #BMK:
	Nr_184		:BOOL;// #MText: #HText: #Prio: #BMK:
	Nr_185		:BOOL;// #MText: #HText: #Prio: #BMK:
	Nr_186		:BOOL;// #MText: #HText: #Prio: #BMK:
	Nr_187		:BOOL;// #MText: #HText: #Prio: #BMK:
	Nr_188		:BOOL;// #MText: #HText: #Prio: #BMK:
	Nr_189		:BOOL;// #MText: #HText: #Prio: #BMK:
	Nr_190		:BOOL;// #MText: #HText: #Prio: #BMK:
	Nr_191		:BOOL;// #MText: #HText: #Prio: #BMK:
	Nr_192		:BOOL;// #MText: #HText: #Prio: #BMK:
	Nr_193		:BOOL;// #MText: #HText: #Prio: #BMK:
	Nr_194		:BOOL;// #MText: #HText: #Prio: #BMK:
	Nr_195		:BOOL;// #MText: #HText: #Prio: #BMK:
	Nr_196		:BOOL;// #MText: #HText: #Prio: #BMK:
	Nr_197		:BOOL;// #MText: #HText: #Prio: #BMK:
	Nr_198		:BOOL;// #MText: #HText: #Prio: #BMK:
	Nr_199		:BOOL;// #MText: #HText: #Prio: #BMK:
	
END_STRUCT
END_TYPE

// ---- SRT_Allgemein/0010_Bausteine_mitDuts/DUTs/Meldungen/DUT_Meldungen_4000.TcDUT
TYPE DUT_Meldungen_4000 :
STRUCT
					  // #MText: Achtung ein Fehler #HText: Achtung eine Hilfe #Prio: 1-10 Error 11-20 Warnung 21-30 Info #BMK:	

	Nr_001		:BOOL;// #MText: #HText: #Prio: #BMK:
	Nr_002		:BOOL;// #MText: #HText: #Prio: #BMK: 
	Nr_003		:BOOL;// #MText: #HText: #Prio: #BMK: 
	Nr_004		:BOOL;// #MText: #HText: #Prio: #BMK: 
	Nr_005		:BOOL;// #MText: #HText: #Prio: #BMK: 
	Nr_006		:BOOL;// #MText: #HText: #Prio: #BMK: 
	Nr_007		:BOOL;// #MText: #HText: #Prio: #BMK: 
	Nr_008		:BOOL;// #MText: #HText: #Prio: #BMK: 
	Nr_009		:BOOL;// #MText: #HText: #Prio: #BMK: 
	Nr_010		:BOOL;// #MText: #HText: #Prio: #BMK: 
	Nr_011		:BOOL;// #MText: #HText: #Prio: #BMK: 
	Nr_012		:BOOL;// #MText: #HText: #Prio: #BMK: 
	Nr_013		:BOOL;// #MText: #HText: #Prio: #BMK: 
	Nr_014		:BOOL;// #MText: #HText: #Prio: #BMK: 
	Nr_015		:BOOL;// #MText: #HText: #Prio: #BMK:     
	Nr_016		:BOOL;// #MText: #HText: #Prio: #BMK:
	Nr_017		:BOOL;// #MText: #HText: #Prio: #BMK:     
	Nr_018		:BOOL;// #MText: #HText: #Prio: #BMK:
	Nr_019		:BOOL;// #MText: #HText: #Prio: #BMK:     
	Nr_020		:BOOL;// #MText: #HText: #Prio: #BMK:
	Nr_021		:BOOL;// #MText: #HText: #Prio: #BMK:     
	Nr_022		:BOOL;// #MText: #HText: #Prio: #BMK:     
	Nr_023		:BOOL;// #MText: #HText: #Prio: #BMK:      
	Nr_024		:BOOL;// #MText: #HText: #Prio: #BMK:
	Nr_025		:BOOL;// #MText: #HText: #Prio: #BMK:      
	Nr_026		:BOOL;// #MText: #HText: #Prio: #BMK:
	Nr_027		:BOOL;// #MText: #HText: #Prio: #BMK:      
	Nr_028		:BOOL;// #MText: #HText: #Prio: #BMK:
	Nr_029		:BOOL;// #MText: #HText: #Prio: #BMK:      
	Nr_030		:BOOL;// #MText: #HText: #Prio: #BMK:
	Nr_031		:BOOL;// #MText: #HText: #Prio: #BMK:      
	Nr_032		:BOOL;// #MText: #HText: #Prio: #BMK:
	Nr_033		:BOOL;// #MText: #HText: #Prio: #BMK:      
	Nr_034		:BOOL;// #MText: #HText: #Prio: #BMK:
	Nr_035		:BOOL;// #MText: #HText: #Prio: #BMK:      
	Nr_036		:BOOL;// #MText: #HText: #Prio: #BMK:
	Nr_037		:BOOL;// #MText: #HText: #Prio: #BMK:
	Nr_038		:BOOL;// #MText: #HText: #Prio: #BMK:
	Nr_039		:BOOL;// #MText: #HText: #Prio: #BMK:
	Nr_040		:BOOL;// #MText: #HText: #Prio: #BMK:
	Nr_041		:BOOL;// #MText: #HText: #Prio: #BMK:
	Nr_042		:BOOL;// #MText: #HText: #Prio: #BMK:
	Nr_043		:BOOL;// #MText: #HText: #Prio: #BMK:
	Nr_044		:BOOL;// #MText: #HText: #Prio: #BMK:
	Nr_045		:BOOL;// #MText: #HText: #Prio: #BMK:
	Nr_046		:BOOL;// #MText: #HText: #Prio: #BMK:
	Nr_047		:BOOL;// #MText: #HText: #Prio: #BMK:
	Nr_048		:BOOL;// #MText: #HText: #Prio: #BMK:
	Nr_049		:BOOL;// #MText: #HText: #Prio: #BMK:
	Nr_050		:BOOL;// #MText: #HText: #Prio: #BMK:
	Nr_051		:BOOL;// #MText: #HText: #Prio: #BMK:
	Nr_052		:BOOL;// #MText: #HText: #Prio: #BMK:
	Nr_053		:BOOL;// #MText: #HText: #Prio: #BMK:
	Nr_054		:BOOL;// #MText: #HText: #Prio: #BMK:
	Nr_055		:BOOL;// #MText: #HText: #Prio: #BMK:
	Nr_056		:BOOL;// #MText: #HText: #Prio: #BMK:
	Nr_057		:BOOL;// #MText: #HText: #Prio: #BMK:
	Nr_058		:BOOL;// #MText: #HText: #Prio: #BMK:
	Nr_059		:BOOL;// #MText: #HText: #Prio: #BMK:
	Nr_060		:BOOL;// #MText: #HText: #Prio: #BMK:
	Nr_061		:BOOL;// #MText: #HText: #Prio: #BMK:
	Nr_062		:BOOL;// #MText: #HText: #Prio: #BMK:
	Nr_063		:BOOL;// #MText: #HText: #Prio: #BMK:
	Nr_064		:BOOL;// #MText: #HText: #Prio: #BMK:
	Nr_065		:BOOL;// #MText: #HText: #Prio: #BMK:
	Nr_066		:BOOL;// #MText: #HText: #Prio: #BMK:
	Nr_067		:BOOL;// #MText: #HText: #Prio: #BMK:
	Nr_068		:BOOL;// #MText: #HText: #Prio: #BMK:
	Nr_069		:BOOL;// #MText: #HText: #Prio: #BMK:
	Nr_070		:BOOL;// #MText: #HText: #Prio: #BMK:
	Nr_071		:BOOL;// #MText: #HText: #Prio: #BMK:
	Nr_072		:BOOL;// #MText: #HText: #Prio: #BMK:
	Nr_073		:BOOL;// #MText: #HText: #Prio: #BMK:
	Nr_074		:BOOL;// #MText: #HText: #Prio: #BMK:
	Nr_075		:BOOL;// #MText: #HText: #Prio: #BMK:
	Nr_076		:BOOL;// #MText: #HText: #Prio: #BMK:
	Nr_077		:BOOL;// #MText: #HText: #Prio: #BMK:
	Nr_078		:BOOL;// #MText: #HText: #Prio: #BMK:
	Nr_079		:BOOL;// #MText: #HText: #Prio: #BMK:
	Nr_080		:BOOL;// #MText: #HText: #Prio: #BMK:
	Nr_081		:BOOL;// #MText: #HText: #Prio: #BMK:
	Nr_082		:BOOL;// #MText: #HText: #Prio: #BMK:
	Nr_083		:BOOL;// #MText: #HText: #Prio: #BMK:
	Nr_084		:BOOL;// #MText: #HText: #Prio: #BMK:
	Nr_085		:BOOL;// #MText: #HText: #Prio: #BMK:
	Nr_086		:BOOL;// #MText: #HText: #Prio: #BMK:
	Nr_087		:BOOL;// #MText: #HText: #Prio: #BMK:
	Nr_088		:BOOL;// #MText: #HText: #Prio: #BMK:
	Nr_089		:BOOL;// #MText: #HText: #Prio: #BMK:
	Nr_090		:BOOL;// #MText: #HText: #Prio: #BMK:
	Nr_091		:BOOL;// #MText: #HText: #Prio: #BMK:
	Nr_092		:BOOL;// #MText: #HText: #Prio: #BMK:
	Nr_093		:BOOL;// #MText: #HText: #Prio: #BMK:
	Nr_094		:BOOL;// #MText: #HText: #Prio: #BMK:
	Nr_095		:BOOL;// #MText: #HText: #Prio: #BMK:
	Nr_096		:BOOL;// #MText: #HText: #Prio: #BMK:
	Nr_097		:BOOL;// #MText: #HText: #Prio: #BMK:
	Nr_098		:BOOL;// #MText: #HText: #Prio: #BMK:
	Nr_099		:BOOL;// #MText: #HText: #Prio: #BMK:
	
